KUKA KRL program: EPS_2_251806_MH58A_A_20260213065155.src

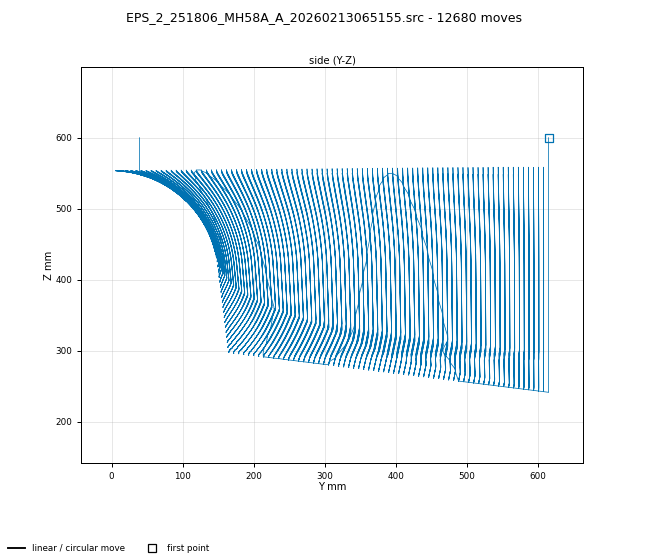
[picture p0: tool path of EPS_2_251806_MH58A_A_20260213065155.src, 12680 of 12682 moves have a stored position in this frame; points joined in program order, loops and branches not executed]
&ACCESS RVP
&REL 4
&COMMENT QRS 19112012
&PARAM EDITMASK = *
DEF PART()
EXT BAS (BAS_COMMAND :IN,REAL :IN )
INT I
BAS (#INITMOV,0 )

;KUKA QRS Post kuka4.cps  Date:22-06-2017 !

File_ID=3039

QRS_PRE_INIT()

;Init var - Until changes are made in qrs_pre_init
Outlet_Square_prg=0
Inlet_1_Square_prg=0
Inlet_2_Square_prg=0
Inlet_3_Square_prg=0
Inlet_4_Square_prg=0
Inlet_5_Square_prg=0

Outlet_1={X 0.000, Y 532.860, Z 433.000, B 0.000, E1 0.000 }
Inlet_1={X 0.000, Y 533.580, Z 423.000, B 0.000, E1 180.000 }
Outlet_1_type=251
Inlet_1_type=251
;QRS#1=Sidecore dimensions
;QRS#2=250-10" PVC SDR 35
;QRS#3=250-10" PVC SDR 35
;QRS#4=
;QRS#5=
;QRS#6=
;QRS#7=
;QRS#8=
;QRS#9=14M PSX
;QRS#10=14M PSX
;QRS#11=
;QRS#12=
;QRS#13=
;QRS#14=
;QRS#15=
;QRS#16=1220x127x838 2,75'
;QRS#17=EPS Height
;QRS#18=558,5
;QRS#19=*
;QRS#20= UPDATED VERSION 22-06-2017
;QRS#21=*
Outlet_Square=0100
Inlet_1_Square=0100
Inlet_2_Square=0
Inlet_3_Square=0
Inlet_4_Square=0
Inlet_5_Square=0
Mill_Square=1
Outlet_Square_Prg=205
Inlet_1_Square_prg=205

QRS_INIT()

$ADVANCE=5

; T1
PTP {E1 173.6,E2 173.6}
PTP {X 0,Y 615.5,A -85,B 0,C 180,E1 173.6,E2 173.6,E3 0,E4 0,E5 0,E6 0}
QRS_SPEED_INIT()
LIN {X 0,Y 615.5,Z 600,A -85,B 0,C 180,E1 173.6,E2 173.6,E3 0,E4 0,E5 0,E6 0} C_VEL
LIN {X 0,Y 615.5,Z 251.488,A -85,B 0,C 180,E1 173.6,E2 173.6} C_VEL
LIN {X 0,Y 615.5,Z 243.309,A -85,B 0,C 180,E1 173.6,E2 173.6} C_VEL
LIN {X 0,Y 615.485,Z 241.309,A -85,B 0,C 180,E1 173.413,E2 173.413} C_VEL
LIN {X 0,Y 615.489,Z 241.322,A -85,B 0,C 180,E1 170.801,E2 170.801} C_VEL
LIN {X 0,Y 615.477,Z 241.314,A -85,B 0,C 180,E1 168.139,E2 168.139} C_VEL
LIN {X 0,Y 615.482,Z 241.311,A -85,B 0,C 180,E1 165.451,E2 165.451} C_VEL
LIN {X 0,Y 615.491,Z 241.324,A -85,B 0,C 180,E1 162.73,E2 162.73} C_VEL
LIN {X 0,Y 615.489,Z 241.307,A -85,B 0,C 180,E1 159.967,E2 159.967} C_VEL
LIN {X 0,Y 615.482,Z 241.32,A -85,B 0,C 180,E1 157.155,E2 157.155} C_VEL
LIN {X 0,Y 615.476,Z 241.315,A -85,B 0,C 180,E1 154.431,E2 154.431} C_VEL
LIN {X 0,Y 615.483,Z 241.309,A -85,B 0,C 180,E1 152.085,E2 152.085} C_VEL
LIN {X 0,Y 615.488,Z 241.308,A -85,B 0,C 180,E1 149.84,E2 149.84} C_VEL
LIN {X 0,Y 615.478,Z 241.316,A -85,B 0,C 180,E1 147.542,E2 147.542} C_VEL
LIN {X 0,Y 615.494,Z 241.324,A -85,B 0,C 180,E1 145.185,E2 145.185} C_VEL
LIN {X 0,Y 615.476,Z 241.317,A -85,B 0,C 180,E1 142.757,E2 142.757} C_VEL
LIN {X 0,Y 615.484,Z 241.31,A -85,B 0,C 180,E1 139.91,E2 139.91} C_VEL
LIN {X 0,Y 615.481,Z 241.317,A -85,B 0,C 180,E1 137.646,E2 137.646} C_VEL
LIN {X 0,Y 615.477,Z 241.318,A -85,B 0,C 180,E1 134.93,E2 134.93} C_VEL
LIN {X 0,Y 615.486,Z 241.31,A -85,B 0,C 180,E1 132.08,E2 132.08} C_VEL
LIN {X 0,Y 615.482,Z 241.318,A -85,B 0,C 180,E1 129.75,E2 129.75} C_VEL
LIN {X 0,Y 615.474,Z 241.315,A -85,B 0,C 180,E1 126.935,E2 126.935} C_VEL
LIN {X 0,Y 615.48,Z 241.31,A -85,B 0,C 180,E1 124.699,E2 124.699} C_VEL
LIN {X 0,Y 615.491,Z 241.308,A -85,B 0,C 180,E1 122.331,E2 122.331} C_VEL
LIN {X 0,Y 615.485,Z 241.322,A -85,B 0,C 180,E1 119.406,E2 119.406} C_VEL
LIN {X 0,Y 615.473,Z 241.314,A -85,B 0,C 180,E1 117.042,E2 117.042} C_VEL
LIN {X 0,Y 615.483,Z 241.312,A -85,B 0,C 180,E1 114.272,E2 114.272} C_VEL
LIN {X 0,Y 615.493,Z 241.527,A -85,B 0,C 180,E1 111.651,E2 111.651} C_VEL
LIN {X 0,Y 615.453,Z 258.15,A -85,B 0,C 180,E1 109.339,E2 109.339} C_VEL
LIN {X 0,Y 615.483,Z 279.634,A -85,B 0,C 180,E1 106.429,E2 106.429} C_VEL
LIN {X 0,Y 615.481,Z 286.32,A -85,B 0,C 180,E1 105.565,E2 105.565} C_VEL
LIN {X 0,Y 615.477,Z 291.213,A -85,B 0,C 180,E1 105.48,E2 105.48} C_VEL
LIN {X 0,Y 615.499,Z 423.163,A -85,B 0,C 180,E1 103.905,E2 103.905} C_VEL
LIN {X 0,Y 615.497,Z 436.757,A -85,B 0,C 180,E1 103.621,E2 103.621} C_VEL
LIN {X 0,Y 615.498,Z 450.494,A -85,B 0,C 180,E1 103.201,E2 103.201} C_VEL
LIN {X 0,Y 615.492,Z 462.905,A -85,B 0,C 180,E1 102.697,E2 102.697} C_VEL
LIN {X 0,Y 615.486,Z 475.846,A -85,B 0,C 180,E1 102.028,E2 102.028} C_VEL
LIN {X 0,Y 615.499,Z 487.561,A -85,B 0,C 180,E1 101.276,E2 101.276} C_VEL
LIN {X 0,Y 615.498,Z 499.228,A -85,B 0,C 180,E1 100.36,E2 100.36} C_VEL
LIN {X 0,Y 615.497,Z 509.651,A -85,B 0,C 180,E1 99.364,E2 99.364} C_VEL
LIN {X 0,Y 615.496,Z 518.241,A -85,B 0,C 180,E1 98.371,E2 98.371} C_VEL
LIN {X 0,Y 615.495,Z 526.453,A -85,B 0,C 180,E1 97.215,E2 97.215} C_VEL
LIN {X 0,Y 615.496,Z 532.184,A -85,B 0,C 180,E1 96.227,E2 96.227} C_VEL
LIN {X 0,Y 615.494,Z 536.888,A -85,B 0,C 180,E1 95.241,E2 95.241} C_VEL
LIN {X 0,Y 615.496,Z 541.757,A -85,B 0,C 180,E1 93.928,E2 93.928} C_VEL
LIN {X 0,Y 615.496,Z 545.154,A -85,B 0,C 180,E1 92.618,E2 92.618} C_VEL
LIN {X 0,Y 615.493,Z 547.174,A -85,B 0,C 180,E1 91.309,E2 91.309} C_VEL
LIN {X 0,Y 615.494,Z 547.884,A -85,B 0,C 180,E1 90,E2 90} C_VEL
LIN {X 0,Y 615.49,Z 547.28,A -85,B 0,C 180,E1 88.691,E2 88.691} C_VEL
LIN {X 0,Y 615.493,Z 545.351,A -85,B 0,C 180,E1 87.382,E2 87.382} C_VEL
LIN {X 0,Y 615.496,Z 542.046,A -85,B 0,C 180,E1 86.072,E2 86.072} C_VEL
LIN {X 0,Y 615.496,Z 537.274,A -85,B 0,C 180,E1 84.759,E2 84.759} C_VEL
LIN {X 0,Y 615.494,Z 530.875,A -85,B 0,C 180,E1 83.444,E2 83.444} C_VEL
LIN {X 0,Y 615.496,Z 523.745,A -85,B 0,C 180,E1 82.29,E2 82.29} C_VEL
LIN {X 0,Y 615.497,Z 516.273,A -85,B 0,C 180,E1 81.298,E2 81.298} C_VEL
LIN {X 0,Y 615.496,Z 507.294,A -85,B 0,C 180,E1 80.304,E2 80.304} C_VEL
LIN {X 0,Y 615.499,Z 496.207,A -85,B 0,C 180,E1 79.291,E2 79.291} C_VEL
LIN {X 0,Y 615.498,Z 485.285,A -85,B 0,C 180,E1 78.474,E2 78.474} C_VEL
LIN {X 0,Y 615.486,Z 472.989,A -85,B 0,C 180,E1 77.721,E2 77.721} C_VEL
LIN {X 0,Y 615.494,Z 461.152,A -85,B 0,C 180,E1 77.135,E2 77.135} C_VEL
LIN {X 0,Y 615.495,Z 448.228,A -85,B 0,C 180,E1 76.631,E2 76.631} C_VEL
LIN {X 0,Y 615.498,Z 435.252,A -85,B 0,C 180,E1 76.253,E2 76.253} C_VEL
LIN {X 0,Y 615.497,Z 421.994,A -85,B 0,C 180,E1 75.988,E2 75.988} C_VEL
LIN {X 0,Y 615.477,Z 286.866,A -85,B 0,C 180,E1 74.371,E2 74.371} C_VEL
LIN {X 0,Y 615.483,Z 285.51,A -85,B 0,C 180,E1 74.265,E2 74.265} C_VEL
LIN {X 0,Y 615.476,Z 265.395,A -85,B 0,C 180,E1 71.558,E2 71.558} C_VEL
LIN {X 0,Y 615.499,Z 243.55,A -85,B 0,C 180,E1 68.569,E2 68.569} C_VEL
LIN {X 0,Y 615.497,Z 241.424,A -85,B 0,C 180,E1 68.217,E2 68.217} C_VEL
LIN {X 0,Y 615.486,Z 241.313,A -85,B 0,C 180,E1 65.729,E2 65.729} C_VEL
LIN {X 0,Y 615.468,Z 241.314,A -85,B 0,C 180,E1 62.959,E2 62.959} C_VEL
LIN {X 0,Y 615.491,Z 241.323,A -85,B 0,C 180,E1 60.205,E2 60.205} C_VEL
LIN {X 0,Y 615.493,Z 241.307,A -85,B 0,C 180,E1 57.544,E2 57.544} C_VEL
LIN {X 0,Y 615.473,Z 241.312,A -85,B 0,C 180,E1 55.185,E2 55.185} C_VEL
LIN {X 0,Y 615.477,Z 241.32,A -85,B 0,C 180,E1 52.758,E2 52.758} C_VEL
LIN {X 0,Y 615.484,Z 241.311,A -85,B 0,C 180,E1 49.912,E2 49.912} C_VEL
LIN {X 0,Y 615.495,Z 241.306,A -85,B 0,C 180,E1 47.649,E2 47.649} C_VEL
LIN {X 0,Y 615.475,Z 241.32,A -85,B 0,C 180,E1 44.932,E2 44.932} C_VEL
LIN {X 0,Y 615.485,Z 241.312,A -85,B 0,C 180,E1 42.081,E2 42.081} C_VEL
LIN {X 0,Y 615.489,Z 241.307,A -85,B 0,C 180,E1 39.75,E2 39.75} C_VEL
LIN {X 0,Y 615.477,Z 241.324,A -85,B 0,C 180,E1 36.937,E2 36.937} C_VEL
LIN {X 0,Y 615.488,Z 241.308,A -85,B 0,C 180,E1 34.022,E2 34.022} C_VEL
LIN {X 0,Y 615.48,Z 241.322,A -85,B 0,C 180,E1 31.087,E2 31.087} C_VEL
LIN {X 0,Y 615.482,Z 241.315,A -85,B 0,C 180,E1 28.452,E2 28.452} C_VEL
LIN {X 0,Y 615.476,Z 241.311,A -85,B 0,C 180,E1 25.716,E2 25.716} C_VEL
LIN {X 0,Y 615.473,Z 241.315,A -85,B 0,C 180,E1 23.557,E2 23.557} C_VEL
LIN {X 0,Y 615.476,Z 241.318,A -85,B 0,C 180,E1 21.432,E2 21.432} C_VEL
LIN {X 0,Y 615.481,Z 241.314,A -85,B 0,C 180,E1 18.607,E2 18.607} C_VEL
LIN {X 0,Y 615.477,Z 241.311,A -85,B 0,C 180,E1 15.906,E2 15.906} C_VEL
LIN {X 0,Y 615.497,Z 241.326,A -85,B 0,C 180,E1 13.201,E2 13.201} C_VEL
LIN {X 0,Y 615.487,Z 241.309,A -85,B 0,C 180,E1 10.527,E2 10.527} C_VEL
LIN {X 0,Y 615.475,Z 241.314,A -85,B 0,C 180,E1 7.876,E2 7.876} C_VEL
LIN {X 0,Y 615.491,Z 241.323,A -85,B 0,C 180,E1 5.241,E2 5.241} C_VEL
LIN {X 0,Y 615.489,Z 241.308,A -85,B 0,C 180,E1 2.618,E2 2.618} C_VEL
LIN {X 0,Y 615.476,Z 241.315,A -85,B 0,C 180,E1 0,E2 0} C_VEL
LIN {X 0,Y 615.49,Z 241.322,A -85,B 0,C 180,E1 -2.618,E2 -2.618} C_VEL
LIN {X 0,Y 615.488,Z 241.308,A -85,B 0,C 180,E1 -5.241,E2 -5.241} C_VEL
LIN {X 0,Y 615.477,Z 241.315,A -85,B 0,C 180,E1 -7.876,E2 -7.876} C_VEL
LIN {X 0,Y 615.487,Z 241.321,A -85,B 0,C 180,E1 -10.527,E2 -10.527} C_VEL
LIN {X 0,Y 615.494,Z 241.306,A -85,B 0,C 180,E1 -13.201,E2 -13.201} C_VEL
LIN {X 0,Y 615.477,Z 241.319,A -85,B 0,C 180,E1 -15.905,E2 -15.905} C_VEL
LIN {X 0,Y 615.476,Z 241.316,A -85,B 0,C 180,E1 -18.646,E2 -18.646} C_VEL
LIN {X 0,Y 615.479,Z 241.311,A -85,B 0,C 180,E1 -21.432,E2 -21.432} C_VEL
LIN {X 0,Y 615.482,Z 241.322,A -85,B 0,C 180,E1 -24.272,E2 -24.272} C_VEL
LIN {X 0,Y 615.49,Z 241.307,A -85,B 0,C 180,E1 -27.177,E2 -27.177} C_VEL
LIN {X 0,Y 615.486,Z 241.321,A -85,B 0,C 180,E1 -30.16,E2 -30.16} C_VEL
LIN {X 0,Y 615.473,Z 241.315,A -85,B 0,C 180,E1 -32.458,E2 -32.458} C_VEL
LIN {X 0,Y 615.49,Z 241.307,A -85,B 0,C 180,E1 -34.815,E2 -34.815} C_VEL
LIN {X 0,Y 615.481,Z 241.313,A -85,B 0,C 180,E1 -37.243,E2 -37.243} C_VEL
LIN {X 0,Y 615.479,Z 241.319,A -85,B 0,C 180,E1 -40.09,E2 -40.09} C_VEL
LIN {X 0,Y 615.475,Z 241.313,A -85,B 0,C 180,E1 -42.354,E2 -42.354} C_VEL
LIN {X 0,Y 615.482,Z 241.312,A -85,B 0,C 180,E1 -45.069,E2 -45.069} C_VEL
LIN {X 0,Y 615.48,Z 241.32,A -85,B 0,C 180,E1 -47.921,E2 -47.921} C_VEL
LIN {X 0,Y 615.475,Z 241.313,A -85,B 0,C 180,E1 -50.25,E2 -50.25} C_VEL
LIN {X 0,Y 615.479,Z 241.315,A -85,B 0,C 180,E1 -53.065,E2 -53.065} C_VEL
LIN {X 0,Y 615.488,Z 241.321,A -85,B 0,C 180,E1 -55.299,E2 -55.299} C_VEL
LIN {X 0,Y 615.483,Z 241.321,A -85,B 0,C 180,E1 -57.67,E2 -57.67} C_VEL
LIN {X 0,Y 615.493,Z 241.307,A -85,B 0,C 180,E1 -60.595,E2 -60.595} C_VEL
LIN {X 0,Y 615.481,Z 241.322,A -85,B 0,C 180,E1 -63.556,E2 -63.556} C_VEL
LIN {X 0,Y 615.486,Z 241.308,A -85,B 0,C 180,E1 -66.444,E2 -66.444} C_VEL
LIN {X 0,Y 615.497,Z 241.502,A -85,B 0,C 180,E1 -67.343,E2 -67.343} C_VEL
LIN {X 0,Y 615.494,Z 249.16,A -85,B 0,C 180,E1 -68.393,E2 -68.393} C_VEL
LIN {X 0,Y 615.433,Z 270.63,A -85,B 0,C 180,E1 -71.18,E2 -71.18} C_VEL
LIN {X 0,Y 615.481,Z 291.387,A -85,B 0,C 180,E1 -73.838,E2 -73.838} C_VEL
LIN {X 0,Y 615.49,Z 296.026,A -85,B 0,C 180,E1 -74.393,E2 -74.393} C_VEL
LIN {X 0,Y 615.479,Z 315.746,A -85,B 0,C 180,E1 -74.647,E2 -74.647} C_VEL
LIN {X 0,Y 615.5,Z 433.901,A -85,B 0,C 180,E1 -76.063,E2 -76.063} C_VEL
LIN {X 0,Y 615.497,Z 448.389,A -85,B 0,C 180,E1 -76.379,E2 -76.379} C_VEL
LIN {X 0,Y 615.496,Z 461.697,A -85,B 0,C 180,E1 -76.799,E2 -76.799} C_VEL
LIN {X 0,Y 615.497,Z 473.843,A -85,B 0,C 180,E1 -77.303,E2 -77.303} C_VEL
LIN {X 0,Y 615.485,Z 486.605,A -85,B 0,C 180,E1 -77.972,E2 -77.972} C_VEL
LIN {X 0,Y 615.499,Z 499.344,A -85,B 0,C 180,E1 -78.807,E2 -78.807} C_VEL
LIN {X 0,Y 615.498,Z 509.751,A -85,B 0,C 180,E1 -79.64,E2 -79.64} C_VEL
LIN {X 0,Y 615.496,Z 520.09,A -85,B 0,C 180,E1 -80.636,E2 -80.636} C_VEL
LIN {X 0,Y 615.497,Z 528.604,A -85,B 0,C 180,E1 -81.629,E2 -81.629} C_VEL
LIN {X 0,Y 615.496,Z 536.728,A -85,B 0,C 180,E1 -82.785,E2 -82.785} C_VEL
LIN {X 0,Y 615.496,Z 542.431,A -85,B 0,C 180,E1 -83.773,E2 -83.773} C_VEL
LIN {X 0,Y 615.495,Z 547.081,A -85,B 0,C 180,E1 -84.759,E2 -84.759} C_VEL
LIN {X 0,Y 615.494,Z 551.902,A -85,B 0,C 180,E1 -86.072,E2 -86.072} C_VEL
LIN {X 0,Y 615.496,Z 555.252,A -85,B 0,C 180,E1 -87.382,E2 -87.382} C_VEL
LIN {X 0,Y 615.489,Z 557.229,A -85,B 0,C 180,E1 -88.691,E2 -88.691} C_VEL
LIN {X 0,Y 615.493,Z 557.889,A -85,B 0,C 180,E1 -90,E2 -90} C_VEL
LIN {X 0,Y 615.489,Z 557.229,A -85,B 0,C 180,E1 -91.309,E2 -91.309} C_VEL
LIN {X 0,Y 615.496,Z 555.252,A -85,B 0,C 180,E1 -92.618,E2 -92.618} C_VEL
LIN {X 0,Y 615.494,Z 551.902,A -85,B 0,C 180,E1 -93.928,E2 -93.928} C_VEL
LIN {X 0,Y 615.495,Z 547.081,A -85,B 0,C 180,E1 -95.241,E2 -95.241} C_VEL
LIN {X 0,Y 615.496,Z 540.628,A -85,B 0,C 180,E1 -96.556,E2 -96.556} C_VEL
LIN {X 0,Y 615.497,Z 533.441,A -85,B 0,C 180,E1 -97.71,E2 -97.71} C_VEL
LIN {X 0,Y 615.498,Z 525.904,A -85,B 0,C 180,E1 -98.702,E2 -98.702} C_VEL
LIN {X 0,Y 615.496,Z 516.854,A -85,B 0,C 180,E1 -99.696,E2 -99.696} C_VEL
LIN {X 0,Y 615.498,Z 506.758,A -85,B 0,C 180,E1 -100.618,E2 -100.618} C_VEL
LIN {X 0,Y 615.498,Z 495.86,A -85,B 0,C 180,E1 -101.443,E2 -101.443} C_VEL
LIN {X 0,Y 615.485,Z 483.71,A -85,B 0,C 180,E1 -102.195,E2 -102.195} C_VEL
LIN {X 0,Y 615.495,Z 470.095,A -85,B 0,C 180,E1 -102.865,E2 -102.865} C_VEL
LIN {X 0,Y 615.496,Z 456.841,A -85,B 0,C 180,E1 -103.369,E2 -103.369} C_VEL
LIN {X 0,Y 615.498,Z 443.296,A -85,B 0,C 180,E1 -103.747,E2 -103.747} C_VEL
LIN {X 0,Y 615.497,Z 428.756,A -85,B 0,C 180,E1 -104.013,E2 -104.013} C_VEL
LIN {X 0,Y 615.488,Z 296.53,A -85,B 0,C 180,E1 -105.586,E2 -105.586} C_VEL
LIN {X 0,Y 615.493,Z 295.48,A -85,B 0,C 180,E1 -105.65,E2 -105.65} C_VEL
LIN {X 0,Y 615.435,Z 273.652,A -85,B 0,C 180,E1 -108.431,E2 -108.431} C_VEL
LIN {X 0,Y 615.46,Z 254.529,A -85,B 0,C 180,E1 -110.906,E2 -110.906} C_VEL
LIN {X 0,Y 615.497,Z 241.605,A -85,B 0,C 180,E1 -112.626,E2 -112.626} C_VEL
LIN {X 0,Y 615.492,Z 241.323,A -85,B 0,C 180,E1 -112.844,E2 -112.844} C_VEL
LIN {X 0,Y 615.485,Z 241.308,A -85,B 0,C 180,E1 -115.715,E2 -115.715} C_VEL
LIN {X 0,Y 615.486,Z 241.327,A -85,B 0,C 180,E1 -118.657,E2 -118.657} C_VEL
LIN {X 0,Y 615.482,Z 241.314,A -85,B 0,C 180,E1 -121.085,E2 -121.085} C_VEL
LIN {X 0,Y 615.492,Z 241.307,A -85,B 0,C 180,E1 -123.535,E2 -123.535} C_VEL
LIN {X 0,Y 615.482,Z 241.327,A -85,B 0,C 180,E1 -126.424,E2 -126.424} C_VEL
LIN {X 0,Y 615.484,Z 241.311,A -85,B 0,C 180,E1 -129.062,E2 -129.062} C_VEL
LIN {X 0,Y 615.486,Z 241.308,A -85,B 0,C 180,E1 -131.473,E2 -131.473} C_VEL
LIN {X 0,Y 615.485,Z 241.321,A -85,B 0,C 180,E1 -134.149,E2 -134.149} C_VEL
LIN {X 0,Y 615.484,Z 241.311,A -85,B 0,C 180,E1 -136.952,E2 -136.952} C_VEL
LIN {X 0,Y 615.48,Z 241.31,A -85,B 0,C 180,E1 -139.393,E2 -139.393} C_VEL
LIN {X 0,Y 615.483,Z 241.321,A -85,B 0,C 180,E1 -141.987,E2 -141.987} C_VEL
LIN {X 0,Y 615.486,Z 241.32,A -85,B 0,C 180,E1 -144.384,E2 -144.384} C_VEL
LIN {X 0,Y 615.483,Z 241.311,A -85,B 0,C 180,E1 -146.763,E2 -146.763} C_VEL
LIN {X 0,Y 615.486,Z 241.308,A -85,B 0,C 180,E1 -149.08,E2 -149.08} C_VEL
LIN {X 0,Y 615.475,Z 241.316,A -85,B 0,C 180,E1 -151.55,E2 -151.55} C_VEL
LIN {X 0,Y 615.482,Z 241.319,A -85,B 0,C 180,E1 -154.284,E2 -154.284} C_VEL
LIN {X 0,Y 615.478,Z 241.315,A -85,B 0,C 180,E1 -156.443,E2 -156.443} C_VEL
LIN {X 0,Y 615.479,Z 241.312,A -85,B 0,C 180,E1 -158.568,E2 -158.568} C_VEL
LIN {X 0,Y 615.475,Z 241.316,A -85,B 0,C 180,E1 -161.354,E2 -161.354} C_VEL
LIN {X 0,Y 615.482,Z 241.319,A -85,B 0,C 180,E1 -164.095,E2 -164.095} C_VEL
LIN {X 0,Y 615.493,Z 241.306,A -85,B 0,C 180,E1 -166.799,E2 -166.799} C_VEL
LIN {X 0,Y 615.484,Z 241.321,A -85,B 0,C 180,E1 -169.473,E2 -169.473} C_VEL
LIN {X 0,Y 615.478,Z 241.315,A -85,B 0,C 180,E1 -172.124,E2 -172.124} C_VEL
LIN {X 0,Y 615.487,Z 241.308,A -85,B 0,C 180,E1 -174.759,E2 -174.759} C_VEL
LIN {X 0,Y 615.487,Z 241.322,A -85,B 0,C 180,E1 -177.382,E2 -177.382} C_VEL
LIN {X 0,Y 615.478,Z 241.315,A -85,B 0,C 180,E1 -180,E2 -180} C_VEL
LIN {X 0,Y 615.488,Z 241.308,A -85,B 0,C 180,E1 -182.618,E2 -182.618} C_VEL
LIN {X 0,Y 615.487,Z 241.322,A -85,B 0,C 180,E1 -185.241,E2 -185.241} C_VEL
LIN {X 0,Y 615.485,Z 241.309,A -85,B 0,C 180,E1 -186.587,E2 -186.587} C_VEL
LIN {X 0,Y 614.81,Z 241.47,A -85,B 0,C 180,E1 -187.133,E2 -187.133} C_VEL
LIN {X 0,Y 611.978,Z 241.874,A -85,B 0,C 180,E1 -188.019,E2 -188.019} C_VEL
LIN {X 0,Y 609.586,Z 242.191,A -85,B 0,C 180,E1 -188.731,E2 -188.731} C_VEL
LIN {X 0,Y 608.548,Z 242.311,A -85,B 0,C 180,E1 -189.281,E2 -189.281} C_VEL
LIN {X 0,Y 608.457,Z 242.319,A -85,B 0,C 180,E1 -189.467,E2 -189.467} C_VEL
LIN {X 0,Y 608.454,Z 242.313,A -85,B 0,C 180,E1 -192,E2 -192} C_VEL
LIN {X 0,Y 608.472,Z 242.312,A -85,B 0,C 180,E1 -194.721,E2 -194.721} C_VEL
LIN {X 0,Y 608.453,Z 242.318,A -85,B 0,C 180,E1 -197.477,E2 -197.477} C_VEL
LIN {X 0,Y 608.46,Z 242.311,A -85,B 0,C 180,E1 -200.274,E2 -200.274} C_VEL
LIN {X 0,Y 608.449,Z 242.314,A -85,B 0,C 180,E1 -202.477,E2 -202.477} C_VEL
LIN {X 0,Y 608.456,Z 242.315,A -85,B 0,C 180,E1 -204.571,E2 -204.571} C_VEL
LIN {X 0,Y 608.48,Z 242.316,A -85,B 0,C 180,E1 -207.21,E2 -207.21} C_VEL
LIN {X 0,Y 608.466,Z 242.311,A -85,B 0,C 180,E1 -209.973,E2 -209.973} C_VEL
LIN {X 0,Y 608.454,Z 242.316,A -85,B 0,C 180,E1 -212.523,E2 -212.523} C_VEL
LIN {X 0,Y 608.442,Z 242.317,A -85,B 0,C 180,E1 -215.278,E2 -215.278} C_VEL
LIN {X 0,Y 608.465,Z 242.311,A -85,B 0,C 180,E1 -217.747,E2 -217.747} C_VEL
LIN {X 0,Y 608.449,Z 242.316,A -85,B 0,C 180,E1 -220.33,E2 -220.33} C_VEL
LIN {X 0,Y 608.446,Z 242.32,A -85,B 0,C 180,E1 -222.961,E2 -222.961} C_VEL
LIN {X 0,Y 608.459,Z 242.312,A -85,B 0,C 180,E1 -225.736,E2 -225.736} C_VEL
LIN {X 0,Y 608.463,Z 242.321,A -85,B 0,C 180,E1 -228.658,E2 -228.658} C_VEL
LIN {X 0,Y 608.461,Z 242.311,A -85,B 0,C 180,E1 -231.412,E2 -231.412} C_VEL
LIN {X 0,Y 608.475,Z 242.312,A -85,B 0,C 180,E1 -233.951,E2 -233.951} C_VEL
LIN {X 0,Y 608.469,Z 242.318,A -85,B 0,C 180,E1 -236.33,E2 -236.33} C_VEL
LIN {X 0,Y 608.444,Z 242.319,A -85,B 0,C 180,E1 -238.733,E2 -238.733} C_VEL
LIN {X 0,Y 608.473,Z 242.31,A -85,B 0,C 180,E1 -241.381,E2 -241.381} C_VEL
LIN {X 0,Y 608.478,Z 242.319,A -85,B 0,C 180,E1 -244.278,E2 -244.278} C_VEL
LIN {X 0,Y 608.446,Z 242.316,A -85,B 0,C 180,E1 -246.876,E2 -246.876} C_VEL
LIN {X 0,Y 608.512,Z 242.509,A -85,B 0,C 180,E1 -248.244,E2 -248.244} C_VEL
LIN {X 0,Y 608.516,Z 258.17,A -85,B 0,C 180,E1 -250.432,E2 -250.432} C_VEL
LIN {X 0,Y 608.527,Z 278.525,A -85,B 0,C 180,E1 -253.218,E2 -253.218} C_VEL
LIN {X 0,Y 608.535,Z 286.323,A -85,B 0,C 180,E1 -254.253,E2 -254.253} C_VEL
LIN {X 0,Y 608.651,Z 289.47,A -85,B 0,C 180,E1 -254.32,E2 -254.32} C_VEL
LIN {X 0,Y 608.608,Z 423.991,A -85,B 0,C 180,E1 -255.949,E2 -255.949} C_VEL
LIN {X 0,Y 608.613,Z 438.305,A -85,B 0,C 180,E1 -256.264,E2 -256.264} C_VEL
LIN {X 0,Y 608.586,Z 451.65,A -85,B 0,C 180,E1 -256.689,E2 -256.689} C_VEL
LIN {X 0,Y 608.542,Z 464.709,A -85,B 0,C 180,E1 -257.24,E2 -257.24} C_VEL
LIN {X 0,Y 608.529,Z 477.345,A -85,B 0,C 180,E1 -257.917,E2 -257.917} C_VEL
LIN {X 0,Y 608.499,Z 488.854,A -85,B 0,C 180,E1 -258.677,E2 -258.677} C_VEL
LIN {X 0,Y 608.495,Z 499.414,A -85,B 0,C 180,E1 -259.519,E2 -259.519} C_VEL
LIN {X 0,Y 608.48,Z 509.9,A -85,B 0,C 180,E1 -260.527,E2 -260.527} C_VEL
LIN {X 0,Y 608.463,Z 518.552,A -85,B 0,C 180,E1 -261.532,E2 -261.532} C_VEL
LIN {X 0,Y 608.46,Z 526.84,A -85,B 0,C 180,E1 -262.701,E2 -262.701} C_VEL
LIN {X 0,Y 608.443,Z 533.325,A -85,B 0,C 180,E1 -263.831,E2 -263.831} C_VEL
LIN {X 0,Y 608.435,Z 538.788,A -85,B 0,C 180,E1 -265.03,E2 -265.03} C_VEL
LIN {X 0,Y 608.434,Z 542.298,A -85,B 0,C 180,E1 -266.026,E2 -266.026} C_VEL
LIN {X 0,Y 608.424,Z 545.734,A -85,B 0,C 180,E1 -267.352,E2 -267.352} C_VEL
LIN {X 0,Y 608.446,Z 547.777,A -85,B 0,C 180,E1 -268.676,E2 -268.676} C_VEL
LIN {X 0,Y 608.434,Z 548.495,A -85,B 0,C 180,E1 -270,E2 -270} C_VEL
LIN {X 0,Y 608.443,Z 547.882,A -85,B 0,C 180,E1 -271.324,E2 -271.324} C_VEL
LIN {X 0,Y 608.421,Z 545.928,A -85,B 0,C 180,E1 -272.648,E2 -272.648} C_VEL
LIN {X 0,Y 608.434,Z 542.585,A -85,B 0,C 180,E1 -273.974,E2 -273.974} C_VEL
LIN {X 0,Y 608.44,Z 537.761,A -85,B 0,C 180,E1 -275.302,E2 -275.302} C_VEL
LIN {X 0,Y 608.442,Z 531.474,A -85,B 0,C 180,E1 -276.6,E2 -276.6} C_VEL
LIN {X 0,Y 608.453,Z 524.101,A -85,B 0,C 180,E1 -277.8,E2 -277.8} C_VEL
LIN {X 0,Y 608.476,Z 516.565,A -85,B 0,C 180,E1 -278.803,E2 -278.803} C_VEL
LIN {X 0,Y 608.488,Z 507.52,A -85,B 0,C 180,E1 -279.809,E2 -279.809} C_VEL
LIN {X 0,Y 608.507,Z 496.723,A -85,B 0,C 180,E1 -280.804,E2 -280.804} C_VEL
LIN {X 0,Y 608.523,Z 485.387,A -85,B 0,C 180,E1 -281.66,E2 -281.66} C_VEL
LIN {X 0,Y 608.539,Z 473.045,A -85,B 0,C 180,E1 -282.421,E2 -282.421} C_VEL
LIN {X 0,Y 608.559,Z 461.177,A -85,B 0,C 180,E1 -283.014,E2 -283.014} C_VEL
LIN {X 0,Y 608.581,Z 448.228,A -85,B 0,C 180,E1 -283.524,E2 -283.524} C_VEL
LIN {X 0,Y 608.594,Z 433.992,A -85,B 0,C 180,E1 -283.935,E2 -283.935} C_VEL
LIN {X 0,Y 608.624,Z 419.126,A -85,B 0,C 180,E1 -284.214,E2 -284.214} C_VEL
LIN {X 0,Y 608.565,Z 286.83,A -85,B 0,C 180,E1 -285.811,E2 -285.811} C_VEL
LIN {X 0,Y 608.493,Z 285.56,A -85,B 0,C 180,E1 -285.92,E2 -285.92} C_VEL
LIN {X 0,Y 608.503,Z 266.614,A -85,B 0,C 180,E1 -288.497,E2 -288.497} C_VEL
LIN {X 0,Y 608.579,Z 244.822,A -85,B 0,C 180,E1 -291.509,E2 -291.509} C_VEL
LIN {X 0,Y 608.479,Z 242.468,A -85,B 0,C 180,E1 -291.869,E2 -291.869} C_VEL
LIN {X 0,Y 608.448,Z 242.313,A -85,B 0,C 180,E1 -294.571,E2 -294.571} C_VEL
LIN {X 0,Y 608.464,Z 242.314,A -85,B 0,C 180,E1 -297.204,E2 -297.204} C_VEL
LIN {X 0,Y 608.469,Z 242.316,A -85,B 0,C 180,E1 -299.971,E2 -299.971} C_VEL
LIN {X 0,Y 608.454,Z 242.313,A -85,B 0,C 180,E1 -302.879,E2 -302.879} C_VEL
LIN {X 0,Y 608.441,Z 242.319,A -85,B 0,C 180,E1 -305.277,E2 -305.277} C_VEL
LIN {X 0,Y 608.464,Z 242.312,A -85,B 0,C 180,E1 -308.24,E2 -308.24} C_VEL
LIN {X 0,Y 608.447,Z 242.313,A -85,B 0,C 180,E1 -310.328,E2 -310.328} C_VEL
LIN {X 0,Y 608.443,Z 242.316,A -85,B 0,C 180,E1 -312.959,E2 -312.959} C_VEL
LIN {X 0,Y 608.452,Z 242.317,A -85,B 0,C 180,E1 -315.735,E2 -315.735} C_VEL
LIN {X 0,Y 608.451,Z 242.313,A -85,B 0,C 180,E1 -318.657,E2 -318.657} C_VEL
LIN {X 0,Y 608.466,Z 242.319,A -85,B 0,C 180,E1 -321.412,E2 -321.412} C_VEL
LIN {X 0,Y 608.474,Z 242.31,A -85,B 0,C 180,E1 -323.949,E2 -323.949} C_VEL
LIN {X 0,Y 608.456,Z 242.312,A -85,B 0,C 180,E1 -326.329,E2 -326.329} C_VEL
LIN {X 0,Y 608.47,Z 242.314,A -85,B 0,C 180,E1 -328.727,E2 -328.727} C_VEL
LIN {X 0,Y 608.47,Z 242.316,A -85,B 0,C 180,E1 -331.378,E2 -331.378} C_VEL
LIN {X 0,Y 608.438,Z 242.314,A -85,B 0,C 180,E1 -333.964,E2 -333.964} C_VEL
LIN {X 0,Y 608.466,Z 242.311,A -85,B 0,C 180,E1 -336.155,E2 -336.155} C_VEL
LIN {X 0,Y 608.449,Z 242.322,A -85,B 0,C 180,E1 -339.018,E2 -339.018} C_VEL
LIN {X 0,Y 608.444,Z 242.313,A -85,B 0,C 180,E1 -341.828,E2 -341.828} C_VEL
LIN {X 0,Y 608.471,Z 242.316,A -85,B 0,C 180,E1 -344.594,E2 -344.594} C_VEL
LIN {X 0,Y 608.476,Z 242.312,A -85,B 0,C 180,E1 -347.323,E2 -347.323} C_VEL
LIN {X 0,Y 608.447,Z 242.314,A -85,B 0,C 180,E1 -350.022,E2 -350.022} C_VEL
LIN {X 0,Y 608.478,Z 242.32,A -85,B 0,C 180,E1 -352.701,E2 -352.701} C_VEL
LIN {X 0,Y 608.455,Z 242.313,A -85,B 0,C 180,E1 -355.362,E2 -355.362} C_VEL
LIN {X 0,Y 608.446,Z 242.315,A -85,B 0,C 180,E1 -358.014,E2 -358.014} C_VEL
LIN {X 0,Y 608.479,Z 242.317,A -85,B 0,C 180,E1 -360.662,E2 -360.662} C_VEL
LIN {X 0,Y 608.476,Z 242.31,A -85,B 0,C 180,E1 -363.311,E2 -363.311} C_VEL
LIN {X 0,Y 608.451,Z 242.316,A -85,B 0,C 180,E1 -365.967,E2 -365.967} C_VEL
LIN {X 0,Y 608.455,Z 242.318,A -85,B 0,C 180,E1 -368.636,E2 -368.636} C_VEL
LIN {X 0,Y 608.472,Z 242.31,A -85,B 0,C 180,E1 -371.324,E2 -371.324} C_VEL
LIN {X 0,Y 608.458,Z 242.318,A -85,B 0,C 180,E1 -374.038,E2 -374.038} C_VEL
LIN {X 0,Y 608.47,Z 242.312,A -85,B 0,C 180,E1 -376.784,E2 -376.784} C_VEL
LIN {X 0,Y 608.453,Z 242.314,A -85,B 0,C 180,E1 -379.571,E2 -379.571} C_VEL
LIN {X 0,Y 608.448,Z 242.317,A -85,B 0,C 180,E1 -382.477,E2 -382.477} C_VEL
LIN {X 0,Y 608.452,Z 242.315,A -85,B 0,C 180,E1 -384.571,E2 -384.571} C_VEL
LIN {X 0,Y 608.482,Z 242.309,A -85,B 0,C 180,E1 -387.21,E2 -387.21} C_VEL
LIN {X 0,Y 608.467,Z 242.322,A -85,B 0,C 180,E1 -389.974,E2 -389.974} C_VEL
LIN {X 0,Y 608.449,Z 242.314,A -85,B 0,C 180,E1 -392.523,E2 -392.523} C_VEL
LIN {X 0,Y 608.443,Z 242.315,A -85,B 0,C 180,E1 -395.278,E2 -395.278} C_VEL
LIN {X 0,Y 608.465,Z 242.32,A -85,B 0,C 180,E1 -397.747,E2 -397.747} C_VEL
LIN {X 0,Y 608.445,Z 242.315,A -85,B 0,C 180,E1 -400.33,E2 -400.33} C_VEL
LIN {X 0,Y 608.468,Z 242.314,A -85,B 0,C 180,E1 -403.31,E2 -403.31} C_VEL
LIN {X 0,Y 608.465,Z 242.314,A -85,B 0,C 180,E1 -406.131,E2 -406.131} C_VEL
LIN {X 0,Y 608.456,Z 242.312,A -85,B 0,C 180,E1 -408.825,E2 -408.825} C_VEL
LIN {X 0,Y 608.463,Z 242.319,A -85,B 0,C 180,E1 -411.413,E2 -411.413} C_VEL
LIN {X 0,Y 608.442,Z 242.317,A -85,B 0,C 180,E1 -413.955,E2 -413.955} C_VEL
LIN {X 0,Y 608.464,Z 242.311,A -85,B 0,C 180,E1 -416.33,E2 -416.33} C_VEL
LIN {X 0,Y 608.475,Z 242.311,A -85,B 0,C 180,E1 -418.728,E2 -418.728} C_VEL
LIN {X 0,Y 608.472,Z 242.321,A -85,B 0,C 180,E1 -421.38,E2 -421.38} C_VEL
LIN {X 0,Y 608.474,Z 242.31,A -85,B 0,C 180,E1 -424.279,E2 -424.279} C_VEL
LIN {X 0,Y 608.5,Z 242.427,A -85,B 0,C 180,E1 -427.193,E2 -427.193} C_VEL
LIN {X 0,Y 608.596,Z 245.132,A -85,B 0,C 180,E1 -427.6,E2 -427.6} C_VEL
LIN {X 0,Y 608.545,Z 267.959,A -85,B 0,C 180,E1 -430.608,E2 -430.608} C_VEL
LIN {X 0,Y 608.453,Z 288.1,A -85,B 0,C 180,E1 -433.216,E2 -433.216} C_VEL
LIN {X 0,Y 608.551,Z 296.02,A -85,B 0,C 180,E1 -434.21,E2 -434.21} C_VEL
LIN {X 0,Y 608.669,Z 299.648,A -85,B 0,C 180,E1 -434.278,E2 -434.278} C_VEL
LIN {X 0,Y 608.621,Z 432.931,A -85,B 0,C 180,E1 -435.885,E2 -435.885} C_VEL
LIN {X 0,Y 608.607,Z 446.874,A -85,B 0,C 180,E1 -436.179,E2 -436.179} C_VEL
LIN {X 0,Y 608.565,Z 460.597,A -85,B 0,C 180,E1 -436.604,E2 -436.604} C_VEL
LIN {X 0,Y 608.562,Z 473.889,A -85,B 0,C 180,E1 -437.156,E2 -437.156} C_VEL
LIN {X 0,Y 608.513,Z 486.685,A -85,B 0,C 180,E1 -437.832,E2 -437.832} C_VEL
LIN {X 0,Y 608.499,Z 499.474,A -85,B 0,C 180,E1 -438.677,E2 -438.677} C_VEL
LIN {X 0,Y 608.496,Z 509.934,A -85,B 0,C 180,E1 -439.519,E2 -439.519} C_VEL
LIN {X 0,Y 608.479,Z 520.336,A -85,B 0,C 180,E1 -440.527,E2 -440.527} C_VEL
LIN {X 0,Y 608.464,Z 528.916,A -85,B 0,C 180,E1 -441.532,E2 -441.532} C_VEL
LIN {X 0,Y 608.461,Z 537.115,A -85,B 0,C 180,E1 -442.701,E2 -442.701} C_VEL
LIN {X 0,Y 608.444,Z 543.546,A -85,B 0,C 180,E1 -443.831,E2 -443.831} C_VEL
LIN {X 0,Y 608.437,Z 548.962,A -85,B 0,C 180,E1 -445.03,E2 -445.03} C_VEL
LIN {X 0,Y 608.431,Z 552.442,A -85,B 0,C 180,E1 -446.026,E2 -446.026} C_VEL
LIN {X 0,Y 608.424,Z 555.831,A -85,B 0,C 180,E1 -447.352,E2 -447.352} C_VEL
LIN {X 0,Y 608.442,Z 557.83,A -85,B 0,C 180,E1 -448.676,E2 -448.676} C_VEL
LIN {X 0,Y 608.433,Z 558.5,A -85,B 0,C 180,E1 -450,E2 -450} C_VEL
LIN {X 0,Y 608.442,Z 557.83,A -85,B 0,C 180,E1 -451.324,E2 -451.324} C_VEL
LIN {X 0,Y 608.424,Z 555.831,A -85,B 0,C 180,E1 -452.648,E2 -452.648} C_VEL
LIN {X 0,Y 608.431,Z 552.441,A -85,B 0,C 180,E1 -453.974,E2 -453.974} C_VEL
LIN {X 0,Y 608.44,Z 547.568,A -85,B 0,C 180,E1 -455.302,E2 -455.302} C_VEL
LIN {X 0,Y 608.445,Z 541.212,A -85,B 0,C 180,E1 -456.603,E2 -456.603} C_VEL
LIN {X 0,Y 608.453,Z 533.798,A -85,B 0,C 180,E1 -457.8,E2 -457.8} C_VEL
LIN {X 0,Y 608.473,Z 524.824,A -85,B 0,C 180,E1 -458.97,E2 -458.97} C_VEL
LIN {X 0,Y 608.473,Z 515.392,A -85,B 0,C 180,E1 -459.977,E2 -459.977} C_VEL
LIN {X 0,Y 608.506,Z 504.047,A -85,B 0,C 180,E1 -460.973,E2 -460.973} C_VEL
LIN {X 0,Y 608.531,Z 492.151,A -85,B 0,C 180,E1 -461.829,E2 -461.829} C_VEL
LIN {X 0,Y 608.529,Z 479.076,A -85,B 0,C 180,E1 -462.591,E2 -462.591} C_VEL
LIN {X 0,Y 608.561,Z 466.177,A -85,B 0,C 180,E1 -463.184,E2 -463.184} C_VEL
LIN {X 0,Y 608.596,Z 452.189,A -85,B 0,C 180,E1 -463.672,E2 -463.672} C_VEL
LIN {X 0,Y 608.621,Z 438.464,A -85,B 0,C 180,E1 -464.012,E2 -464.012} C_VEL
LIN {X 0,Y 608.627,Z 422.183,A -85,B 0,C 180,E1 -464.257,E2 -464.257} C_VEL
LIN {X 0,Y 608.604,Z 296.517,A -85,B 0,C 180,E1 -465.767,E2 -465.767} C_VEL
LIN {X 0,Y 608.521,Z 295.525,A -85,B 0,C 180,E1 -465.834,E2 -465.834} C_VEL
LIN {X 0,Y 608.48,Z 274.9,A -85,B 0,C 180,E1 -468.489,E2 -468.489} C_VEL
LIN {X 0,Y 608.518,Z 257.4,A -85,B 0,C 180,E1 -470.778,E2 -470.778} C_VEL
LIN {X 0,Y 608.561,Z 242.969,A -85,B 0,C 180,E1 -472.697,E2 -472.697} C_VEL
LIN {X 0,Y 608.487,Z 242.382,A -85,B 0,C 180,E1 -472.852,E2 -472.852} C_VEL
LIN {X 0,Y 608.474,Z 242.31,A -85,B 0,C 180,E1 -475.721,E2 -475.721} C_VEL
LIN {X 0,Y 608.472,Z 242.321,A -85,B 0,C 180,E1 -478.62,E2 -478.62} C_VEL
LIN {X 0,Y 608.458,Z 242.313,A -85,B 0,C 180,E1 -481.316,E2 -481.316} C_VEL
LIN {X 0,Y 608.472,Z 242.31,A -85,B 0,C 180,E1 -483.735,E2 -483.735} C_VEL
LIN {X 0,Y 608.442,Z 242.318,A -85,B 0,C 180,E1 -486.092,E2 -486.092} C_VEL
LIN {X 0,Y 608.463,Z 242.319,A -85,B 0,C 180,E1 -488.587,E2 -488.587} C_VEL
LIN {X 0,Y 608.462,Z 242.311,A -85,B 0,C 180,E1 -491.342,E2 -491.342} C_VEL
LIN {X 0,Y 608.453,Z 242.322,A -85,B 0,C 180,E1 -494.264,E2 -494.264} C_VEL
LIN {X 0,Y 608.45,Z 242.313,A -85,B 0,C 180,E1 -497.04,E2 -497.04} C_VEL
LIN {X 0,Y 608.446,Z 242.315,A -85,B 0,C 180,E1 -499.696,E2 -499.696} C_VEL
LIN {X 0,Y 608.465,Z 242.321,A -85,B 0,C 180,E1 -502.253,E2 -502.253} C_VEL
LIN {X 0,Y 608.479,Z 242.308,A -85,B 0,C 180,E1 -505.089,E2 -505.089} C_VEL
LIN {X 0,Y 608.458,Z 242.319,A -85,B 0,C 180,E1 -507.905,E2 -507.905} C_VEL
LIN {X 0,Y 608.473,Z 242.317,A -85,B 0,C 180,E1 -510.221,E2 -510.221} C_VEL
LIN {X 0,Y 608.45,Z 242.313,A -85,B 0,C 180,E1 -513.226,E2 -513.226} C_VEL
LIN {X 0,Y 608.47,Z 242.317,A -85,B 0,C 180,E1 -516.155,E2 -516.155} C_VEL
LIN {X 0,Y 608.447,Z 242.313,A -85,B 0,C 180,E1 -519.018,E2 -519.018} C_VEL
LIN {X 0,Y 608.445,Z 242.324,A -85,B 0,C 180,E1 -521.828,E2 -521.828} C_VEL
LIN {X 0,Y 608.471,Z 242.31,A -85,B 0,C 180,E1 -524.594,E2 -524.594} C_VEL
LIN {X 0,Y 608.473,Z 242.314,A -85,B 0,C 180,E1 -527.323,E2 -527.323} C_VEL
LIN {X 0,Y 608.45,Z 242.318,A -85,B 0,C 180,E1 -530.023,E2 -530.023} C_VEL
LIN {X 0,Y 608.477,Z 242.309,A -85,B 0,C 180,E1 -532.701,E2 -532.701} C_VEL
LIN {X 0,Y 608.451,Z 242.319,A -85,B 0,C 180,E1 -535.362,E2 -535.362} C_VEL
LIN {X 0,Y 608.449,Z 242.316,A -85,B 0,C 180,E1 -538.014,E2 -538.014} C_VEL
LIN {X 0,Y 608.476,Z 242.31,A -85,B 0,C 180,E1 -540.662,E2 -540.662} C_VEL
LIN {X 0,Y 608.476,Z 242.317,A -85,B 0,C 180,E1 -543.311,E2 -543.311} C_VEL
LIN {X 0,Y 608.452,Z 242.314,A -85,B 0,C 180,E1 -545.967,E2 -545.967} C_VEL
LIN {X 0,Y 608.455,Z 242.313,A -85,B 0,C 180,E1 -548.636,E2 -548.636} C_VEL
LIN {X 0,Y 608.457,Z 242.319,A -85,B 0,C 180,E1 -549.467,E2 -549.467} C_VEL
LIN {X 0,Y 607.773,Z 242.399,A -85,B 0,C 180,E1 -550.02,E2 -550.02} C_VEL
LIN {X 0,Y 604.915,Z 242.757,A -85,B 0,C 180,E1 -550.917,E2 -550.917} C_VEL
LIN {X 0,Y 602.513,Z 243.057,A -85,B 0,C 180,E1 -551.638,E2 -551.638} C_VEL
LIN {X 0,Y 601.487,Z 243.181,A -85,B 0,C 180,E1 -552.195,E2 -552.195} C_VEL
LIN {X 0,Y 601.405,Z 243.19,A -85,B 0,C 180,E1 -552.383,E2 -552.383} C_VEL
LIN {X 0,Y 601.426,Z 243.192,A -85,B 0,C 180,E1 -554.897,E2 -554.897} C_VEL
LIN {X 0,Y 601.427,Z 243.194,A -85,B 0,C 180,E1 -556.986,E2 -556.986} C_VEL
LIN {X 0,Y 601.405,Z 243.191,A -85,B 0,C 180,E1 -559.81,E2 -559.81} C_VEL
LIN {X 0,Y 601.404,Z 243.194,A -85,B 0,C 180,E1 -562.683,E2 -562.683} C_VEL
LIN {X 0,Y 601.402,Z 243.198,A -85,B 0,C 180,E1 -564.879,E2 -564.879} C_VEL
LIN {X 0,Y 601.417,Z 243.189,A -85,B 0,C 180,E1 -567.868,E2 -567.868} C_VEL
LIN {X 0,Y 601.442,Z 243.186,A -85,B 0,C 180,E1 -570.163,E2 -570.163} C_VEL
LIN {X 0,Y 601.415,Z 243.195,A -85,B 0,C 180,E1 -572.716,E2 -572.716} C_VEL
LIN {X 0,Y 601.412,Z 243.195,A -85,B 0,C 180,E1 -575.116,E2 -575.116} C_VEL
LIN {X 0,Y 601.429,Z 243.189,A -85,B 0,C 180,E1 -577.42,E2 -577.42} C_VEL
LIN {X 0,Y 601.408,Z 243.19,A -85,B 0,C 180,E1 -579.996,E2 -579.996} C_VEL
LIN {X 0,Y 601.406,Z 243.199,A -85,B 0,C 180,E1 -582.671,E2 -582.671} C_VEL
LIN {X 0,Y 601.422,Z 243.189,A -85,B 0,C 180,E1 -585.483,E2 -585.483} C_VEL
LIN {X 0,Y 601.424,Z 243.194,A -85,B 0,C 180,E1 -588.407,E2 -588.407} C_VEL
LIN {X 0,Y 601.409,Z 243.195,A -85,B 0,C 180,E1 -590.874,E2 -590.874} C_VEL
LIN {X 0,Y 601.44,Z 243.187,A -85,B 0,C 180,E1 -593.735,E2 -593.735} C_VEL
LIN {X 0,Y 601.429,Z 243.194,A -85,B 0,C 180,E1 -596.687,E2 -596.687} C_VEL
LIN {X 0,Y 601.41,Z 243.191,A -85,B 0,C 180,E1 -599.058,E2 -599.058} C_VEL
LIN {X 0,Y 601.432,Z 243.186,A -85,B 0,C 180,E1 -601.374,E2 -601.374} C_VEL
LIN {X 0,Y 601.418,Z 243.196,A -85,B 0,C 180,E1 -604.132,E2 -604.132} C_VEL
LIN {X 0,Y 601.417,Z 243.197,A -85,B 0,C 180,E1 -606.59,E2 -606.59} C_VEL
LIN {X 0,Y 601.471,Z 243.338,A -85,B 0,C 180,E1 -608.089,E2 -608.089} C_VEL
LIN {X 0,Y 601.637,Z 251.494,A -85,B 0,C 180,E1 -609.262,E2 -609.262} C_VEL
LIN {X 0,Y 601.533,Z 270.896,A -85,B 0,C 180,E1 -611.965,E2 -611.965} C_VEL
LIN {X 0,Y 601.519,Z 286.324,A -85,B 0,C 180,E1 -614.064,E2 -614.064} C_VEL
LIN {X 0,Y 601.828,Z 289.515,A -85,B 0,C 180,E1 -614.138,E2 -614.138} C_VEL
LIN {X 0,Y 601.731,Z 423.063,A -85,B 0,C 180,E1 -615.767,E2 -615.767} C_VEL
LIN {X 0,Y 601.712,Z 437.51,A -85,B 0,C 180,E1 -616.081,E2 -616.081} C_VEL
LIN {X 0,Y 601.673,Z 450.539,A -85,B 0,C 180,E1 -616.49,E2 -616.49} C_VEL
LIN {X 0,Y 601.632,Z 462.965,A -85,B 0,C 180,E1 -617.005,E2 -617.005} C_VEL
LIN {X 0,Y 601.561,Z 475.945,A -85,B 0,C 180,E1 -617.689,E2 -617.689} C_VEL
LIN {X 0,Y 601.513,Z 487.703,A -85,B 0,C 180,E1 -618.458,E2 -618.458} C_VEL
LIN {X 0,Y 601.481,Z 499.422,A -85,B 0,C 180,E1 -619.396,E2 -619.396} C_VEL
LIN {X 0,Y 601.431,Z 509.905,A -85,B 0,C 180,E1 -620.415,E2 -620.415} C_VEL
LIN {X 0,Y 601.406,Z 518.556,A -85,B 0,C 180,E1 -621.431,E2 -621.431} C_VEL
LIN {X 0,Y 601.391,Z 526.843,A -85,B 0,C 180,E1 -622.614,E2 -622.614} C_VEL
LIN {X 0,Y 601.361,Z 532.512,A -85,B 0,C 180,E1 -623.605,E2 -623.605} C_VEL
LIN {X 0,Y 601.354,Z 537.378,A -85,B 0,C 180,E1 -624.635,E2 -624.635} C_VEL
LIN {X 0,Y 601.345,Z 542.3,A -85,B 0,C 180,E1 -625.979,E2 -625.979} C_VEL
LIN {X 0,Y 601.324,Z 545.735,A -85,B 0,C 180,E1 -627.32,E2 -627.32} C_VEL
LIN {X 0,Y 601.346,Z 547.779,A -85,B 0,C 180,E1 -628.661,E2 -628.661} C_VEL
LIN {X 0,Y 601.334,Z 548.496,A -85,B 0,C 180,E1 -630,E2 -630} C_VEL
LIN {X 0,Y 601.343,Z 547.882,A -85,B 0,C 180,E1 -631.339,E2 -631.339} C_VEL
LIN {X 0,Y 601.321,Z 545.927,A -85,B 0,C 180,E1 -632.679,E2 -632.679} C_VEL
LIN {X 0,Y 601.346,Z 542.584,A -85,B 0,C 180,E1 -634.021,E2 -634.021} C_VEL
LIN {X 0,Y 601.355,Z 537.759,A -85,B 0,C 180,E1 -635.365,E2 -635.365} C_VEL
LIN {X 0,Y 601.368,Z 531.889,A -85,B 0,C 180,E1 -636.601,E2 -636.601} C_VEL
LIN {X 0,Y 601.386,Z 525.219,A -85,B 0,C 180,E1 -637.723,E2 -637.723} C_VEL
LIN {X 0,Y 601.411,Z 516.561,A -85,B 0,C 180,E1 -638.907,E2 -638.907} C_VEL
LIN {X 0,Y 601.432,Z 507.514,A -85,B 0,C 180,E1 -639.925,E2 -639.925} C_VEL
LIN {X 0,Y 601.474,Z 496.336,A -85,B 0,C 180,E1 -640.964,E2 -640.964} C_VEL
LIN {X 0,Y 601.542,Z 484.103,A -85,B 0,C 180,E1 -641.883,E2 -641.883} C_VEL
LIN {X 0,Y 601.561,Z 471.471,A -85,B 0,C 180,E1 -642.653,E2 -642.653} C_VEL
LIN {X 0,Y 601.63,Z 459.198,A -85,B 0,C 180,E1 -643.253,E2 -643.253} C_VEL
LIN {X 0,Y 601.697,Z 445.161,A -85,B 0,C 180,E1 -643.783,E2 -643.783} C_VEL
LIN {X 0,Y 601.729,Z 431.543,A -85,B 0,C 180,E1 -644.155,E2 -644.155} C_VEL
LIN {X 0,Y 601.754,Z 417.595,A -85,B 0,C 180,E1 -644.401,E2 -644.401} C_VEL
LIN {X 0,Y 601.671,Z 287.425,A -85,B 0,C 180,E1 -645.983,E2 -645.983} C_VEL
LIN {X 0,Y 601.503,Z 285.909,A -85,B 0,C 180,E1 -646.067,E2 -646.067} C_VEL
LIN {X 0,Y 601.531,Z 267.303,A -85,B 0,C 180,E1 -648.623,E2 -648.623} C_VEL
LIN {X 0,Y 601.667,Z 246.091,A -85,B 0,C 180,E1 -651.589,E2 -651.589} C_VEL
LIN {X 0,Y 601.436,Z 243.277,A -85,B 0,C 180,E1 -652.047,E2 -652.047} C_VEL
LIN {X 0,Y 601.397,Z 243.192,A -85,B 0,C 180,E1 -654.878,E2 -654.878} C_VEL
LIN {X 0,Y 601.42,Z 243.196,A -85,B 0,C 180,E1 -657.867,E2 -657.867} C_VEL
LIN {X 0,Y 601.427,Z 243.191,A -85,B 0,C 180,E1 -660.163,E2 -660.163} C_VEL
LIN {X 0,Y 601.423,Z 243.188,A -85,B 0,C 180,E1 -662.715,E2 -662.715} C_VEL
LIN {X 0,Y 601.393,Z 243.195,A -85,B 0,C 180,E1 -665.111,E2 -665.111} C_VEL
LIN {X 0,Y 601.431,Z 243.196,A -85,B 0,C 180,E1 -667.418,E2 -667.418} C_VEL
LIN {X 0,Y 601.407,Z 243.193,A -85,B 0,C 180,E1 -669.994,E2 -669.994} C_VEL
LIN {X 0,Y 601.409,Z 243.19,A -85,B 0,C 180,E1 -672.669,E2 -672.669} C_VEL
LIN {X 0,Y 601.421,Z 243.197,A -85,B 0,C 180,E1 -675.481,E2 -675.481} C_VEL
LIN {X 0,Y 601.418,Z 243.188,A -85,B 0,C 180,E1 -678.406,E2 -678.406} C_VEL
LIN {X 0,Y 601.429,Z 243.191,A -85,B 0,C 180,E1 -680.875,E2 -680.875} C_VEL
LIN {X 0,Y 601.439,Z 243.189,A -85,B 0,C 180,E1 -683.733,E2 -683.733} C_VEL
LIN {X 0,Y 601.427,Z 243.186,A -85,B 0,C 180,E1 -686.063,E2 -686.063} C_VEL
LIN {X 0,Y 601.434,Z 243.188,A -85,B 0,C 180,E1 -688.541,E2 -688.541} C_VEL
LIN {X 0,Y 601.429,Z 243.193,A -85,B 0,C 180,E1 -691.373,E2 -691.373} C_VEL
LIN {X 0,Y 601.398,Z 243.193,A -85,B 0,C 180,E1 -693.636,E2 -693.636} C_VEL
LIN {X 0,Y 601.416,Z 243.193,A -85,B 0,C 180,E1 -696.589,E2 -696.589} C_VEL
LIN {X 0,Y 601.426,Z 243.19,A -85,B 0,C 180,E1 -699.478,E2 -699.478} C_VEL
LIN {X 0,Y 601.394,Z 243.194,A -85,B 0,C 180,E1 -702.311,E2 -702.311} C_VEL
LIN {X 0,Y 601.414,Z 243.193,A -85,B 0,C 180,E1 -704.409,E2 -704.409} C_VEL
LIN {X 0,Y 601.422,Z 243.192,A -85,B 0,C 180,E1 -707.172,E2 -707.172} C_VEL
LIN {X 0,Y 601.426,Z 243.188,A -85,B 0,C 180,E1 -709.905,E2 -709.905} C_VEL
LIN {X 0,Y 601.446,Z 243.194,A -85,B 0,C 180,E1 -712.615,E2 -712.615} C_VEL
LIN {X 0,Y 601.423,Z 243.189,A -85,B 0,C 180,E1 -715.308,E2 -715.308} C_VEL
LIN {X 0,Y 601.417,Z 243.19,A -85,B 0,C 180,E1 -717.991,E2 -717.991} C_VEL
LIN {X 0,Y 601.449,Z 243.193,A -85,B 0,C 180,E1 -720.669,E2 -720.669} C_VEL
LIN {X 0,Y 601.427,Z 243.187,A -85,B 0,C 180,E1 -723.35,E2 -723.35} C_VEL
LIN {X 0,Y 601.405,Z 243.194,A -85,B 0,C 180,E1 -726.037,E2 -726.037} C_VEL
LIN {X 0,Y 601.434,Z 243.191,A -85,B 0,C 180,E1 -728.738,E2 -728.738} C_VEL
LIN {X 0,Y 601.428,Z 243.187,A -85,B 0,C 180,E1 -731.458,E2 -731.458} C_VEL
LIN {X 0,Y 601.41,Z 243.199,A -85,B 0,C 180,E1 -734.206,E2 -734.206} C_VEL
LIN {X 0,Y 601.427,Z 243.188,A -85,B 0,C 180,E1 -736.986,E2 -736.986} C_VEL
LIN {X 0,Y 601.406,Z 243.195,A -85,B 0,C 180,E1 -739.809,E2 -739.809} C_VEL
LIN {X 0,Y 601.403,Z 243.192,A -85,B 0,C 180,E1 -742.683,E2 -742.683} C_VEL
LIN {X 0,Y 601.4,Z 243.191,A -85,B 0,C 180,E1 -744.879,E2 -744.879} C_VEL
LIN {X 0,Y 601.416,Z 243.197,A -85,B 0,C 180,E1 -747.868,E2 -747.868} C_VEL
LIN {X 0,Y 601.441,Z 243.193,A -85,B 0,C 180,E1 -750.163,E2 -750.163} C_VEL
LIN {X 0,Y 601.412,Z 243.189,A -85,B 0,C 180,E1 -752.716,E2 -752.716} C_VEL
LIN {X 0,Y 601.411,Z 243.189,A -85,B 0,C 180,E1 -755.116,E2 -755.116} C_VEL
LIN {X 0,Y 601.429,Z 243.191,A -85,B 0,C 180,E1 -757.42,E2 -757.42} C_VEL
LIN {X 0,Y 601.406,Z 243.197,A -85,B 0,C 180,E1 -759.996,E2 -759.996} C_VEL
LIN {X 0,Y 601.406,Z 243.19,A -85,B 0,C 180,E1 -762.671,E2 -762.671} C_VEL
LIN {X 0,Y 601.421,Z 243.196,A -85,B 0,C 180,E1 -765.483,E2 -765.483} C_VEL
LIN {X 0,Y 601.422,Z 243.188,A -85,B 0,C 180,E1 -768.407,E2 -768.407} C_VEL
LIN {X 0,Y 601.43,Z 243.188,A -85,B 0,C 180,E1 -770.876,E2 -770.876} C_VEL
LIN {X 0,Y 601.398,Z 243.2,A -85,B 0,C 180,E1 -773.418,E2 -773.418} C_VEL
LIN {X 0,Y 601.431,Z 243.189,A -85,B 0,C 180,E1 -776.065,E2 -776.065} C_VEL
LIN {X 0,Y 601.439,Z 243.186,A -85,B 0,C 180,E1 -778.543,E2 -778.543} C_VEL
LIN {X 0,Y 601.432,Z 243.197,A -85,B 0,C 180,E1 -781.374,E2 -781.374} C_VEL
LIN {X 0,Y 601.4,Z 243.197,A -85,B 0,C 180,E1 -783.637,E2 -783.637} C_VEL
LIN {X 0,Y 601.419,Z 243.193,A -85,B 0,C 180,E1 -786.59,E2 -786.59} C_VEL
LIN {X 0,Y 601.469,Z 243.431,A -85,B 0,C 180,E1 -787.07,E2 -787.07} C_VEL
LIN {X 0,Y 601.697,Z 247.842,A -85,B 0,C 180,E1 -787.694,E2 -787.694} C_VEL
LIN {X 0,Y 601.559,Z 270.644,A -85,B 0,C 180,E1 -790.729,E2 -790.729} C_VEL
LIN {X 0,Y 601.472,Z 289.867,A -85,B 0,C 180,E1 -793.246,E2 -793.246} C_VEL
LIN {X 0,Y 601.564,Z 296.212,A -85,B 0,C 180,E1 -794.033,E2 -794.033} C_VEL
LIN {X 0,Y 601.835,Z 299.648,A -85,B 0,C 180,E1 -794.094,E2 -794.094} C_VEL
LIN {X 0,Y 601.755,Z 432.93,A -85,B 0,C 180,E1 -795.721,E2 -795.721} C_VEL
LIN {X 0,Y 601.715,Z 447.274,A -85,B 0,C 180,E1 -796.029,E2 -796.029} C_VEL
LIN {X 0,Y 601.659,Z 459.926,A -85,B 0,C 180,E1 -796.422,E2 -796.422} C_VEL
LIN {X 0,Y 601.628,Z 472.101,A -85,B 0,C 180,E1 -796.919,E2 -796.919} C_VEL
LIN {X 0,Y 601.551,Z 485.27,A -85,B 0,C 180,E1 -797.604,E2 -797.604} C_VEL
LIN {X 0,Y 601.511,Z 497.154,A -85,B 0,C 180,E1 -798.373,E2 -798.373} C_VEL
LIN {X 0,Y 601.49,Z 507.996,A -85,B 0,C 180,E1 -799.225,E2 -799.225} C_VEL
LIN {X 0,Y 601.422,Z 518.71,A -85,B 0,C 180,E1 -800.245,E2 -800.245} C_VEL
LIN {X 0,Y 601.407,Z 527.56,A -85,B 0,C 180,E1 -801.262,E2 -801.262} C_VEL
LIN {X 0,Y 601.406,Z 536.041,A -85,B 0,C 180,E1 -802.446,E2 -802.446} C_VEL
LIN {X 0,Y 601.361,Z 542.751,A -85,B 0,C 180,E1 -803.604,E2 -803.604} C_VEL
LIN {X 0,Y 601.355,Z 547.568,A -85,B 0,C 180,E1 -804.635,E2 -804.635} C_VEL
LIN {X 0,Y 601.343,Z 552.442,A -85,B 0,C 180,E1 -805.979,E2 -805.979} C_VEL
LIN {X 0,Y 601.324,Z 555.831,A -85,B 0,C 180,E1 -807.321,E2 -807.321} C_VEL
LIN {X 0,Y 601.342,Z 557.831,A -85,B 0,C 180,E1 -808.661,E2 -808.661} C_VEL
LIN {X 0,Y 601.333,Z 558.5,A -85,B 0,C 180,E1 -810,E2 -810} C_VEL
LIN {X 0,Y 601.342,Z 557.831,A -85,B 0,C 180,E1 -811.339,E2 -811.339} C_VEL
LIN {X 0,Y 601.324,Z 555.832,A -85,B 0,C 180,E1 -812.68,E2 -812.68} C_VEL
LIN {X 0,Y 601.343,Z 552.442,A -85,B 0,C 180,E1 -814.021,E2 -814.021} C_VEL
LIN {X 0,Y 601.355,Z 547.568,A -85,B 0,C 180,E1 -815.365,E2 -815.365} C_VEL
LIN {X 0,Y 601.372,Z 541.623,A -85,B 0,C 180,E1 -816.605,E2 -816.605} C_VEL
LIN {X 0,Y 601.386,Z 534.92,A -85,B 0,C 180,E1 -817.723,E2 -817.723} C_VEL
LIN {X 0,Y 601.412,Z 526.199,A -85,B 0,C 180,E1 -818.907,E2 -818.907} C_VEL
LIN {X 0,Y 601.433,Z 517.083,A -85,B 0,C 180,E1 -819.925,E2 -819.925} C_VEL
LIN {X 0,Y 601.497,Z 506.828,A -85,B 0,C 180,E1 -820.877,E2 -820.877} C_VEL
LIN {X 0,Y 601.533,Z 495.973,A -85,B 0,C 180,E1 -821.712,E2 -821.712} C_VEL
LIN {X 0,Y 601.574,Z 483.781,A -85,B 0,C 180,E1 -822.482,E2 -822.482} C_VEL
LIN {X 0,Y 601.628,Z 472.099,A -85,B 0,C 180,E1 -823.081,E2 -823.081} C_VEL
LIN {X 0,Y 601.669,Z 458.945,A -85,B 0,C 180,E1 -823.612,E2 -823.612} C_VEL
LIN {X 0,Y 601.706,Z 445.035,A -85,B 0,C 180,E1 -824.028,E2 -824.028} C_VEL
LIN {X 0,Y 601.732,Z 430.561,A -85,B 0,C 180,E1 -824.314,E2 -824.314} C_VEL
LIN {X 0,Y 601.729,Z 297.205,A -85,B 0,C 180,E1 -825.938,E2 -825.938} C_VEL
LIN {X 0,Y 601.512,Z 295.525,A -85,B 0,C 180,E1 -826.023,E2 -826.023} C_VEL
LIN {X 0,Y 601.518,Z 274.733,A -85,B 0,C 180,E1 -828.733,E2 -828.733} C_VEL
LIN {X 0,Y 601.612,Z 257.777,A -85,B 0,C 180,E1 -830.977,E2 -830.977} C_VEL
LIN {X 0,Y 601.704,Z 245.131,A -85,B 0,C 180,E1 -832.671,E2 -832.671} C_VEL
LIN {X 0,Y 601.463,Z 243.343,A -85,B 0,C 180,E1 -832.953,E2 -832.953} C_VEL
LIN {X 0,Y 601.436,Z 243.187,A -85,B 0,C 180,E1 -835.617,E2 -835.617} C_VEL
LIN {X 0,Y 601.4,Z 243.192,A -85,B 0,C 180,E1 -837.868,E2 -837.868} C_VEL
LIN {X 0,Y 601.425,Z 243.19,A -85,B 0,C 180,E1 -840.163,E2 -840.163} C_VEL
LIN {X 0,Y 601.421,Z 243.196,A -85,B 0,C 180,E1 -842.715,E2 -842.715} C_VEL
LIN {X 0,Y 601.396,Z 243.193,A -85,B 0,C 180,E1 -845.112,E2 -845.112} C_VEL
LIN {X 0,Y 601.431,Z 243.187,A -85,B 0,C 180,E1 -847.418,E2 -847.418} C_VEL
LIN {X 0,Y 601.398,Z 243.195,A -85,B 0,C 180,E1 -849.995,E2 -849.995} C_VEL
LIN {X 0,Y 601.412,Z 243.195,A -85,B 0,C 180,E1 -852.669,E2 -852.669} C_VEL
LIN {X 0,Y 601.421,Z 243.189,A -85,B 0,C 180,E1 -855.481,E2 -855.481} C_VEL
LIN {X 0,Y 601.42,Z 243.196,A -85,B 0,C 180,E1 -858.406,E2 -858.406} C_VEL
LIN {X 0,Y 601.434,Z 243.188,A -85,B 0,C 180,E1 -860.875,E2 -860.875} C_VEL
LIN {X 0,Y 601.439,Z 243.189,A -85,B 0,C 180,E1 -863.733,E2 -863.733} C_VEL
LIN {X 0,Y 601.428,Z 243.196,A -85,B 0,C 180,E1 -866.063,E2 -866.063} C_VEL
LIN {X 0,Y 601.426,Z 243.188,A -85,B 0,C 180,E1 -869.058,E2 -869.058} C_VEL
LIN {X 0,Y 601.424,Z 243.189,A -85,B 0,C 180,E1 -871.373,E2 -871.373} C_VEL
LIN {X 0,Y 601.4,Z 243.195,A -85,B 0,C 180,E1 -873.636,E2 -873.636} C_VEL
LIN {X 0,Y 601.417,Z 243.19,A -85,B 0,C 180,E1 -876.59,E2 -876.59} C_VEL
LIN {X 0,Y 601.424,Z 243.192,A -85,B 0,C 180,E1 -879.478,E2 -879.478} C_VEL
LIN {X 0,Y 601.397,Z 243.194,A -85,B 0,C 180,E1 -882.312,E2 -882.312} C_VEL
LIN {X 0,Y 601.414,Z 243.191,A -85,B 0,C 180,E1 -884.409,E2 -884.409} C_VEL
LIN {X 0,Y 601.42,Z 243.191,A -85,B 0,C 180,E1 -887.172,E2 -887.172} C_VEL
LIN {X 0,Y 601.427,Z 243.194,A -85,B 0,C 180,E1 -889.905,E2 -889.905} C_VEL
LIN {X 0,Y 601.446,Z 243.185,A -85,B 0,C 180,E1 -892.615,E2 -892.615} C_VEL
LIN {X 0,Y 601.419,Z 243.194,A -85,B 0,C 180,E1 -895.308,E2 -895.308} C_VEL
LIN {X 0,Y 601.419,Z 243.192,A -85,B 0,C 180,E1 -897.991,E2 -897.991} C_VEL
LIN {X 0,Y 601.446,Z 243.185,A -85,B 0,C 180,E1 -900.67,E2 -900.67} C_VEL
LIN {X 0,Y 601.427,Z 243.196,A -85,B 0,C 180,E1 -903.35,E2 -903.35} C_VEL
LIN {X 0,Y 601.405,Z 243.192,A -85,B 0,C 180,E1 -906.037,E2 -906.037} C_VEL
LIN {X 0,Y 601.434,Z 243.188,A -85,B 0,C 180,E1 -908.738,E2 -908.738} C_VEL
LIN {X 0,Y 601.428,Z 243.195,A -85,B 0,C 180,E1 -911.458,E2 -911.458} C_VEL
LIN {X 0,Y 601.405,Z 243.19,A -85,B 0,C 180,E1 -912.383,E2 -912.383} C_VEL
LIN {X 0,Y 600.744,Z 243.279,A -85,B 0,C 180,E1 -912.943,E2 -912.943} C_VEL
LIN {X 0,Y 597.894,Z 243.635,A -85,B 0,C 180,E1 -913.85,E2 -913.85} C_VEL
LIN {X 0,Y 595.482,Z 243.936,A -85,B 0,C 180,E1 -914.581,E2 -914.581} C_VEL
LIN {X 0,Y 594.443,Z 244.066,A -85,B 0,C 180,E1 -915.144,E2 -915.144} C_VEL
LIN {X 0,Y 594.358,Z 244.072,A -85,B 0,C 180,E1 -915.335,E2 -915.335} C_VEL
LIN {X 0,Y 594.374,Z 244.067,A -85,B 0,C 180,E1 -917.904,E2 -917.904} C_VEL
LIN {X 0,Y 594.372,Z 244.073,A -85,B 0,C 180,E1 -920.918,E2 -920.918} C_VEL
LIN {X 0,Y 594.387,Z 244.066,A -85,B 0,C 180,E1 -923.704,E2 -923.704} C_VEL
LIN {X 0,Y 594.383,Z 244.069,A -85,B 0,C 180,E1 -926.7,E2 -926.7} C_VEL
LIN {X 0,Y 594.375,Z 244.076,A -85,B 0,C 180,E1 -928.999,E2 -928.999} C_VEL
LIN {X 0,Y 594.386,Z 244.064,A -85,B 0,C 180,E1 -931.646,E2 -931.646} C_VEL
LIN {X 0,Y 594.394,Z 244.067,A -85,B 0,C 180,E1 -934.579,E2 -934.579} C_VEL
LIN {X 0,Y 594.381,Z 244.072,A -85,B 0,C 180,E1 -937.087,E2 -937.087} C_VEL
LIN {X 0,Y 594.372,Z 244.066,A -85,B 0,C 180,E1 -939.775,E2 -939.775} C_VEL
LIN {X 0,Y 594.364,Z 244.07,A -85,B 0,C 180,E1 -942.376,E2 -942.376} C_VEL
LIN {X 0,Y 594.36,Z 244.071,A -85,B 0,C 180,E1 -945.192,E2 -945.192} C_VEL
LIN {X 0,Y 594.369,Z 244.065,A -85,B 0,C 180,E1 -947.626,E2 -947.626} C_VEL
LIN {X 0,Y 594.387,Z 244.071,A -85,B 0,C 180,E1 -950.321,E2 -950.321} C_VEL
LIN {X 0,Y 594.382,Z 244.07,A -85,B 0,C 180,E1 -952.914,E2 -952.914} C_VEL
LIN {X 0,Y 594.381,Z 244.067,A -85,B 0,C 180,E1 -955.862,E2 -955.862} C_VEL
LIN {X 0,Y 594.369,Z 244.074,A -85,B 0,C 180,E1 -958.65,E2 -958.65} C_VEL
LIN {X 0,Y 594.383,Z 244.066,A -85,B 0,C 180,E1 -961.043,E2 -961.043} C_VEL
LIN {X 0,Y 594.391,Z 244.069,A -85,B 0,C 180,E1 -963.977,E2 -963.977} C_VEL
LIN {X 0,Y 594.388,Z 244.075,A -85,B 0,C 180,E1 -966.296,E2 -966.296} C_VEL
LIN {X 0,Y 594.433,Z 244.274,A -85,B 0,C 180,E1 -967.953,E2 -967.953} C_VEL
LIN {X 0,Y 594.72,Z 249.064,A -85,B 0,C 180,E1 -968.662,E2 -968.662} C_VEL
LIN {X 0,Y 594.563,Z 269.628,A -85,B 0,C 180,E1 -971.567,E2 -971.567} C_VEL
LIN {X 0,Y 594.533,Z 286.326,A -85,B 0,C 180,E1 -973.872,E2 -973.872} C_VEL
LIN {X 0,Y 595.016,Z 289.561,A -85,B 0,C 180,E1 -973.951,E2 -973.951} C_VEL
LIN {X 0,Y 594.851,Z 423.83,A -85,B 0,C 180,E1 -975.613,E2 -975.613} C_VEL
LIN {X 0,Y 594.805,Z 438.286,A -85,B 0,C 180,E1 -975.937,E2 -975.937} C_VEL
LIN {X 0,Y 594.754,Z 452.802,A -85,B 0,C 180,E1 -976.417,E2 -976.417} C_VEL
LIN {X 0,Y 594.644,Z 466.485,A -85,B 0,C 180,E1 -977.023,E2 -977.023} C_VEL
LIN {X 0,Y 594.563,Z 478.779,A -85,B 0,C 180,E1 -977.716,E2 -977.716} C_VEL
LIN {X 0,Y 594.528,Z 491.048,A -85,B 0,C 180,E1 -978.569,E2 -978.569} C_VEL
LIN {X 0,Y 594.448,Z 501.362,A -85,B 0,C 180,E1 -979.441,E2 -979.441} C_VEL
LIN {X 0,Y 594.371,Z 511.462,A -85,B 0,C 180,E1 -980.472,E2 -980.472} C_VEL
LIN {X 0,Y 594.324,Z 519.846,A -85,B 0,C 180,E1 -981.5,E2 -981.5} C_VEL
LIN {X 0,Y 594.303,Z 527.86,A -85,B 0,C 180,E1 -982.697,E2 -982.697} C_VEL
LIN {X 0,Y 594.281,Z 534.314,A -85,B 0,C 180,E1 -983.89,E2 -983.89} C_VEL
LIN {X 0,Y 594.235,Z 540.036,A -85,B 0,C 180,E1 -985.251,E2 -985.251} C_VEL
LIN {X 0,Y 594.259,Z 544.199,A -85,B 0,C 180,E1 -986.61,E2 -986.61} C_VEL
LIN {X 0,Y 594.242,Z 546.927,A -85,B 0,C 180,E1 -987.967,E2 -987.967} C_VEL
LIN {X 0,Y 594.235,Z 548.302,A -85,B 0,C 180,E1 -989.322,E2 -989.322} C_VEL
LIN {X 0,Y 594.236,Z 548.356,A -85,B 0,C 180,E1 -990.678,E2 -990.678} C_VEL
LIN {X 0,Y 594.241,Z 547.073,A -85,B 0,C 180,E1 -992.033,E2 -992.033} C_VEL
LIN {X 0,Y 594.259,Z 544.433,A -85,B 0,C 180,E1 -993.39,E2 -993.39} C_VEL
LIN {X 0,Y 594.236,Z 540.363,A -85,B 0,C 180,E1 -994.749,E2 -994.749} C_VEL
LIN {X 0,Y 594.282,Z 534.741,A -85,B 0,C 180,E1 -996.11,E2 -996.11} C_VEL
LIN {X 0,Y 594.303,Z 528.393,A -85,B 0,C 180,E1 -997.303,E2 -997.303} C_VEL
LIN {X 0,Y 594.324,Z 520.497,A -85,B 0,C 180,E1 -998.5,E2 -998.5} C_VEL
LIN {X 0,Y 594.355,Z 512.242,A -85,B 0,C 180,E1 -999.529,E2 -999.529} C_VEL
LIN {X 0,Y 594.449,Z 502.304,A -85,B 0,C 180,E1 -1000.559,E2 -1000.559} C_VEL
LIN {X 0,Y 594.493,Z 491.167,A -85,B 0,C 180,E1 -1001.512,E2 -1001.512} C_VEL
LIN {X 0,Y 594.581,Z 478.834,A -85,B 0,C 180,E1 -1002.371,E2 -1002.371} C_VEL
LIN {X 0,Y 594.665,Z 466.549,A -85,B 0,C 180,E1 -1003.063,E2 -1003.063} C_VEL
LIN {X 0,Y 594.728,Z 452.882,A -85,B 0,C 180,E1 -1003.67,E2 -1003.67} C_VEL
LIN {X 0,Y 594.806,Z 438.47,A -85,B 0,C 180,E1 -1004.147,E2 -1004.147} C_VEL
LIN {X 0,Y 594.871,Z 425.113,A -85,B 0,C 180,E1 -1004.452,E2 -1004.452} C_VEL
LIN {X 0,Y 594.913,Z 398.858,A -85,B 0,C 180,E1 -1004.801,E2 -1004.801} C_VEL
LIN {X 0,Y 594.874,Z 288.496,A -85,B 0,C 180,E1 -1006.156,E2 -1006.156} C_VEL
LIN {X 0,Y 594.535,Z 286.354,A -85,B 0,C 180,E1 -1006.216,E2 -1006.216} C_VEL
LIN {X 0,Y 594.553,Z 268.998,A -85,B 0,C 180,E1 -1008.611,E2 -1008.611} C_VEL
LIN {X 0,Y 594.724,Z 248.632,A -85,B 0,C 180,E1 -1011.489,E2 -1011.489} C_VEL
LIN {X 0,Y 594.416,Z 244.302,A -85,B 0,C 180,E1 -1012.139,E2 -1012.139} C_VEL
LIN {X 0,Y 594.389,Z 244.066,A -85,B 0,C 180,E1 -1014.445,E2 -1014.445} C_VEL
LIN {X 0,Y 594.38,Z 244.066,A -85,B 0,C 180,E1 -1016.699,E2 -1016.699} C_VEL
LIN {X 0,Y 594.381,Z 244.066,A -85,B 0,C 180,E1 -1018.998,E2 -1018.998} C_VEL
LIN {X 0,Y 594.377,Z 244.076,A -85,B 0,C 180,E1 -1021.642,E2 -1021.642} C_VEL
LIN {X 0,Y 594.376,Z 244.066,A -85,B 0,C 180,E1 -1024.579,E2 -1024.579} C_VEL
LIN {X 0,Y 594.38,Z 244.069,A -85,B 0,C 180,E1 -1027.086,E2 -1027.086} C_VEL
LIN {X 0,Y 594.37,Z 244.072,A -85,B 0,C 180,E1 -1029.773,E2 -1029.773} C_VEL
LIN {X 0,Y 594.368,Z 244.066,A -85,B 0,C 180,E1 -1032.374,E2 -1032.374} C_VEL
LIN {X 0,Y 594.359,Z 244.075,A -85,B 0,C 180,E1 -1035.19,E2 -1035.19} C_VEL
LIN {X 0,Y 594.378,Z 244.064,A -85,B 0,C 180,E1 -1038.151,E2 -1038.151} C_VEL
LIN {X 0,Y 594.382,Z 244.074,A -85,B 0,C 180,E1 -1041.195,E2 -1041.195} C_VEL
LIN {X 0,Y 594.391,Z 244.066,A -85,B 0,C 180,E1 -1043.758,E2 -1043.758} C_VEL
LIN {X 0,Y 594.373,Z 244.064,A -85,B 0,C 180,E1 -1046.238,E2 -1046.238} C_VEL
LIN {X 0,Y 594.384,Z 244.067,A -85,B 0,C 180,E1 -1048.65,E2 -1048.65} C_VEL
LIN {X 0,Y 594.378,Z 244.076,A -85,B 0,C 180,E1 -1051.041,E2 -1051.041} C_VEL
LIN {X 0,Y 594.378,Z 244.065,A -85,B 0,C 180,E1 -1053.976,E2 -1053.976} C_VEL
LIN {X 0,Y 594.388,Z 244.066,A -85,B 0,C 180,E1 -1056.296,E2 -1056.296} C_VEL
LIN {X 0,Y 594.397,Z 244.068,A -85,B 0,C 180,E1 -1059.224,E2 -1059.224} C_VEL
LIN {X 0,Y 594.374,Z 244.067,A -85,B 0,C 180,E1 -1062.096,E2 -1062.096} C_VEL
LIN {X 0,Y 594.366,Z 244.068,A -85,B 0,C 180,E1 -1064.219,E2 -1064.219} C_VEL
LIN {X 0,Y 594.369,Z 244.073,A -85,B 0,C 180,E1 -1067.017,E2 -1067.017} C_VEL
LIN {X 0,Y 594.386,Z 244.064,A -85,B 0,C 180,E1 -1069.784,E2 -1069.784} C_VEL
LIN {X 0,Y 594.394,Z 244.071,A -85,B 0,C 180,E1 -1072.527,E2 -1072.527} C_VEL
LIN {X 0,Y 594.392,Z 244.065,A -85,B 0,C 180,E1 -1075.252,E2 -1075.252} C_VEL
LIN {X 0,Y 594.387,Z 244.065,A -85,B 0,C 180,E1 -1077.967,E2 -1077.967} C_VEL
LIN {X 0,Y 594.419,Z 244.068,A -85,B 0,C 180,E1 -1080.677,E2 -1080.677} C_VEL
LIN {X 0,Y 594.378,Z 244.065,A -85,B 0,C 180,E1 -1083.389,E2 -1083.389} C_VEL
LIN {X 0,Y 594.361,Z 244.073,A -85,B 0,C 180,E1 -1086.109,E2 -1086.109} C_VEL
LIN {X 0,Y 594.395,Z 244.066,A -85,B 0,C 180,E1 -1088.842,E2 -1088.842} C_VEL
LIN {X 0,Y 594.386,Z 244.065,A -85,B 0,C 180,E1 -1091.596,E2 -1091.596} C_VEL
LIN {X 0,Y 594.381,Z 244.074,A -85,B 0,C 180,E1 -1094.377,E2 -1094.377} C_VEL
LIN {X 0,Y 594.385,Z 244.064,A -85,B 0,C 180,E1 -1097.193,E2 -1097.193} C_VEL
LIN {X 0,Y 594.372,Z 244.075,A -85,B 0,C 180,E1 -1100.054,E2 -1100.054} C_VEL
LIN {X 0,Y 594.357,Z 244.068,A -85,B 0,C 180,E1 -1102.968,E2 -1102.968} C_VEL
LIN {X 0,Y 594.371,Z 244.067,A -85,B 0,C 180,E1 -1105.193,E2 -1105.193} C_VEL
LIN {X 0,Y 594.376,Z 244.068,A -85,B 0,C 180,E1 -1107.527,E2 -1107.527} C_VEL
LIN {X 0,Y 594.393,Z 244.068,A -85,B 0,C 180,E1 -1110.331,E2 -1110.331} C_VEL
LIN {X 0,Y 594.371,Z 244.065,A -85,B 0,C 180,E1 -1112.951,E2 -1112.951} C_VEL
LIN {X 0,Y 594.378,Z 244.067,A -85,B 0,C 180,E1 -1115.407,E2 -1115.407} C_VEL
LIN {X 0,Y 594.381,Z 244.074,A -85,B 0,C 180,E1 -1117.941,E2 -1117.941} C_VEL
LIN {X 0,Y 594.374,Z 244.066,A -85,B 0,C 180,E1 -1120.823,E2 -1120.823} C_VEL
LIN {X 0,Y 594.361,Z 244.072,A -85,B 0,C 180,E1 -1123.3,E2 -1123.3} C_VEL
LIN {X 0,Y 594.378,Z 244.068,A -85,B 0,C 180,E1 -1126.16,E2 -1126.16} C_VEL
LIN {X 0,Y 594.379,Z 244.064,A -85,B 0,C 180,E1 -1128.537,E2 -1128.537} C_VEL
LIN {X 0,Y 594.382,Z 244.071,A -85,B 0,C 180,E1 -1131.296,E2 -1131.296} C_VEL
LIN {X 0,Y 594.348,Z 244.076,A -85,B 0,C 180,E1 -1133.756,E2 -1133.756} C_VEL
LIN {X 0,Y 594.378,Z 244.066,A -85,B 0,C 180,E1 -1136.24,E2 -1136.24} C_VEL
LIN {X 0,Y 594.388,Z 244.065,A -85,B 0,C 180,E1 -1138.652,E2 -1138.652} C_VEL
LIN {X 0,Y 594.383,Z 244.068,A -85,B 0,C 180,E1 -1141.043,E2 -1141.043} C_VEL
LIN {X 0,Y 594.386,Z 244.067,A -85,B 0,C 180,E1 -1143.978,E2 -1143.978} C_VEL
LIN {X 0,Y 594.388,Z 244.072,A -85,B 0,C 180,E1 -1146.666,E2 -1146.666} C_VEL
LIN {X 0,Y 594.408,Z 244.287,A -85,B 0,C 180,E1 -1146.897,E2 -1146.897} C_VEL
LIN {X 0,Y 594.825,Z 248.252,A -85,B 0,C 180,E1 -1147.478,E2 -1147.478} C_VEL
LIN {X 0,Y 594.652,Z 270.644,A -85,B 0,C 180,E1 -1150.496,E2 -1150.496} C_VEL
LIN {X 0,Y 594.492,Z 289.158,A -85,B 0,C 180,E1 -1152.95,E2 -1152.95} C_VEL
LIN {X 0,Y 594.589,Z 296.203,A -85,B 0,C 180,E1 -1153.84,E2 -1153.84} C_VEL
LIN {X 0,Y 595.032,Z 299.648,A -85,B 0,C 180,E1 -1153.908,E2 -1153.908} C_VEL
LIN {X 0,Y 594.857,Z 433.904,A -85,B 0,C 180,E1 -1155.569,E2 -1155.569} C_VEL
LIN {X 0,Y 594.818,Z 448.156,A -85,B 0,C 180,E1 -1155.889,E2 -1155.889} C_VEL
LIN {X 0,Y 594.729,Z 461.723,A -85,B 0,C 180,E1 -1156.33,E2 -1156.33} C_VEL
LIN {X 0,Y 594.653,Z 475.643,A -85,B 0,C 180,E1 -1156.937,E2 -1156.937} C_VEL
LIN {X 0,Y 594.581,Z 488.101,A -85,B 0,C 180,E1 -1157.629,E2 -1157.629} C_VEL
LIN {X 0,Y 594.524,Z 500.563,A -85,B 0,C 180,E1 -1158.488,E2 -1158.488} C_VEL
LIN {X 0,Y 594.449,Z 511.839,A -85,B 0,C 180,E1 -1159.441,E2 -1159.441} C_VEL
LIN {X 0,Y 594.368,Z 521.852,A -85,B 0,C 180,E1 -1160.472,E2 -1160.472} C_VEL
LIN {X 0,Y 594.324,Z 530.172,A -85,B 0,C 180,E1 -1161.5,E2 -1161.5} C_VEL
LIN {X 0,Y 594.303,Z 538.127,A -85,B 0,C 180,E1 -1162.697,E2 -1162.697} C_VEL
LIN {X 0,Y 594.281,Z 544.528,A -85,B 0,C 180,E1 -1163.89,E2 -1163.89} C_VEL
LIN {X 0,Y 594.237,Z 550.199,A -85,B 0,C 180,E1 -1165.251,E2 -1165.251} C_VEL
LIN {X 0,Y 594.259,Z 554.315,A -85,B 0,C 180,E1 -1166.61,E2 -1166.61} C_VEL
LIN {X 0,Y 594.241,Z 557,A -85,B 0,C 180,E1 -1167.967,E2 -1167.967} C_VEL
LIN {X 0,Y 594.237,Z 558.332,A -85,B 0,C 180,E1 -1169.322,E2 -1169.322} C_VEL
LIN {X 0,Y 594.237,Z 558.332,A -85,B 0,C 180,E1 -1170.678,E2 -1170.678} C_VEL
LIN {X 0,Y 594.242,Z 557,A -85,B 0,C 180,E1 -1172.033,E2 -1172.033} C_VEL
LIN {X 0,Y 594.259,Z 554.316,A -85,B 0,C 180,E1 -1173.39,E2 -1173.39} C_VEL
LIN {X 0,Y 594.237,Z 550.199,A -85,B 0,C 180,E1 -1174.749,E2 -1174.749} C_VEL
LIN {X 0,Y 594.281,Z 544.527,A -85,B 0,C 180,E1 -1176.11,E2 -1176.11} C_VEL
LIN {X 0,Y 594.303,Z 538.126,A -85,B 0,C 180,E1 -1177.303,E2 -1177.303} C_VEL
LIN {X 0,Y 594.324,Z 530.171,A -85,B 0,C 180,E1 -1178.5,E2 -1178.5} C_VEL
LIN {X 0,Y 594.367,Z 521.852,A -85,B 0,C 180,E1 -1179.528,E2 -1179.528} C_VEL
LIN {X 0,Y 594.449,Z 511.838,A -85,B 0,C 180,E1 -1180.559,E2 -1180.559} C_VEL
LIN {X 0,Y 594.523,Z 500.564,A -85,B 0,C 180,E1 -1181.512,E2 -1181.512} C_VEL
LIN {X 0,Y 594.58,Z 488.1,A -85,B 0,C 180,E1 -1182.371,E2 -1182.371} C_VEL
LIN {X 0,Y 594.653,Z 475.642,A -85,B 0,C 180,E1 -1183.063,E2 -1183.063} C_VEL
LIN {X 0,Y 594.743,Z 461.718,A -85,B 0,C 180,E1 -1183.67,E2 -1183.67} C_VEL
LIN {X 0,Y 594.819,Z 448.137,A -85,B 0,C 180,E1 -1184.111,E2 -1184.111} C_VEL
LIN {X 0,Y 594.874,Z 433.898,A -85,B 0,C 180,E1 -1184.43,E2 -1184.43} C_VEL
LIN {X 0,Y 594.856,Z 297.852,A -85,B 0,C 180,E1 -1186.119,E2 -1186.119} C_VEL
LIN {X 0,Y 594.541,Z 295.718,A -85,B 0,C 180,E1 -1186.194,E2 -1186.194} C_VEL
LIN {X 0,Y 594.569,Z 275.435,A -85,B 0,C 180,E1 -1188.867,E2 -1188.867} C_VEL
LIN {X 0,Y 594.699,Z 258.156,A -85,B 0,C 180,E1 -1191.181,E2 -1191.181} C_VEL
LIN {X 0,Y 594.742,Z 246.081,A -85,B 0,C 180,E1 -1192.821,E2 -1192.821} C_VEL
LIN {X 0,Y 594.387,Z 244.163,A -85,B 0,C 180,E1 -1193.15,E2 -1193.15} C_VEL
LIN {X 0,Y 594.373,Z 244.068,A -85,B 0,C 180,E1 -1195.944,E2 -1195.944} C_VEL
LIN {X 0,Y 594.375,Z 244.071,A -85,B 0,C 180,E1 -1198.226,E2 -1198.226} C_VEL
LIN {X 0,Y 594.381,Z 244.073,A -85,B 0,C 180,E1 -1200.559,E2 -1200.559} C_VEL
LIN {X 0,Y 594.377,Z 244.069,A -85,B 0,C 180,E1 -1202.949,E2 -1202.949} C_VEL
LIN {X 0,Y 594.349,Z 244.07,A -85,B 0,C 180,E1 -1205.408,E2 -1205.408} C_VEL
LIN {X 0,Y 594.381,Z 244.067,A -85,B 0,C 180,E1 -1207.94,E2 -1207.94} C_VEL
LIN {X 0,Y 594.377,Z 244.068,A -85,B 0,C 180,E1 -1210.822,E2 -1210.822} C_VEL
LIN {X 0,Y 594.378,Z 244.068,A -85,B 0,C 180,E1 -1213.84,E2 -1213.84} C_VEL
LIN {X 0,Y 594.361,Z 244.072,A -85,B 0,C 180,E1 -1216.7,E2 -1216.7} C_VEL
LIN {X 0,Y 594.364,Z 244.067,A -85,B 0,C 180,E1 -1219.433,E2 -1219.433} C_VEL
LIN {X 0,Y 594.385,Z 244.071,A -85,B 0,C 180,E1 -1222.391,E2 -1222.391} C_VEL
LIN {X 0,Y 594.38,Z 244.065,A -85,B 0,C 180,E1 -1224.671,E2 -1224.671} C_VEL
LIN {X 0,Y 594.371,Z 244.065,A -85,B 0,C 180,E1 -1227.088,E2 -1227.088} C_VEL
LIN {X 0,Y 594.394,Z 244.068,A -85,B 0,C 180,E1 -1229.669,E2 -1229.669} C_VEL
LIN {X 0,Y 594.384,Z 244.067,A -85,B 0,C 180,E1 -1232.54,E2 -1232.54} C_VEL
LIN {X 0,Y 594.372,Z 244.067,A -85,B 0,C 180,E1 -1234.807,E2 -1234.807} C_VEL
LIN {X 0,Y 594.356,Z 244.069,A -85,B 0,C 180,E1 -1237.264,E2 -1237.264} C_VEL
LIN {X 0,Y 594.373,Z 244.076,A -85,B 0,C 180,E1 -1239.946,E2 -1239.946} C_VEL
LIN {X 0,Y 594.385,Z 244.064,A -85,B 0,C 180,E1 -1242.807,E2 -1242.807} C_VEL
LIN {X 0,Y 594.38,Z 244.075,A -85,B 0,C 180,E1 -1245.825,E2 -1245.825} C_VEL
LIN {X 0,Y 594.387,Z 244.065,A -85,B 0,C 180,E1 -1248.404,E2 -1248.404} C_VEL
LIN {X 0,Y 594.394,Z 244.066,A -85,B 0,C 180,E1 -1251.158,E2 -1251.158} C_VEL
LIN {X 0,Y 594.362,Z 244.073,A -85,B 0,C 180,E1 -1253.891,E2 -1253.891} C_VEL
LIN {X 0,Y 594.378,Z 244.065,A -85,B 0,C 180,E1 -1256.611,E2 -1256.611} C_VEL
LIN {X 0,Y 594.417,Z 244.068,A -85,B 0,C 180,E1 -1259.323,E2 -1259.323} C_VEL
LIN {X 0,Y 594.388,Z 244.065,A -85,B 0,C 180,E1 -1262.033,E2 -1262.033} C_VEL
LIN {X 0,Y 594.393,Z 244.065,A -85,B 0,C 180,E1 -1264.748,E2 -1264.748} C_VEL
LIN {X 0,Y 594.394,Z 244.072,A -85,B 0,C 180,E1 -1267.473,E2 -1267.473} C_VEL
LIN {X 0,Y 594.387,Z 244.064,A -85,B 0,C 180,E1 -1270.216,E2 -1270.216} C_VEL
LIN {X 0,Y 594.368,Z 244.072,A -85,B 0,C 180,E1 -1272.983,E2 -1272.983} C_VEL
LIN {X 0,Y 594.358,Z 244.072,A -85,B 0,C 180,E1 -1275.335,E2 -1275.335} C_VEL
LIN {X 0,Y 593.688,Z 244.154,A -85,B 0,C 180,E1 -1275.901,E2 -1275.901} C_VEL
LIN {X 0,Y 590.833,Z 244.511,A -85,B 0,C 180,E1 -1276.819,E2 -1276.819} C_VEL
LIN {X 0,Y 588.427,Z 244.812,A -85,B 0,C 180,E1 -1277.558,E2 -1277.558} C_VEL
LIN {X 0,Y 587.398,Z 244.936,A -85,B 0,C 180,E1 -1278.128,E2 -1278.128} C_VEL
LIN {X 0,Y 587.317,Z 244.946,A -85,B 0,C 180,E1 -1278.321,E2 -1278.321} C_VEL
LIN {X 0,Y 587.321,Z 244.953,A -85,B 0,C 180,E1 -1281.038,E2 -1281.038} C_VEL
LIN {X 0,Y 587.317,Z 244.953,A -85,B 0,C 180,E1 -1283.259,E2 -1283.259} C_VEL
LIN {X 0,Y 587.33,Z 244.946,A -85,B 0,C 180,E1 -1285.517,E2 -1285.517} C_VEL
LIN {X 0,Y 587.342,Z 244.943,A -85,B 0,C 180,E1 -1287.818,E2 -1287.818} C_VEL
LIN {X 0,Y 587.345,Z 244.945,A -85,B 0,C 180,E1 -1290.513,E2 -1290.513} C_VEL
LIN {X 0,Y 587.329,Z 244.943,A -85,B 0,C 180,E1 -1293.397,E2 -1293.397} C_VEL
LIN {X 0,Y 587.352,Z 244.94,A -85,B 0,C 180,E1 -1295.896,E2 -1295.896} C_VEL
LIN {X 0,Y 587.329,Z 244.949,A -85,B 0,C 180,E1 -1298.48,E2 -1298.48} C_VEL
LIN {X 0,Y 587.332,Z 244.945,A -85,B 0,C 180,E1 -1301.158,E2 -1301.158} C_VEL
LIN {X 0,Y 587.322,Z 244.946,A -85,B 0,C 180,E1 -1304.114,E2 -1304.114} C_VEL
LIN {X 0,Y 587.319,Z 244.948,A -85,B 0,C 180,E1 -1306.995,E2 -1306.995} C_VEL
LIN {X 0,Y 587.315,Z 244.946,A -85,B 0,C 180,E1 -1309.747,E2 -1309.747} C_VEL
LIN {X 0,Y 587.342,Z 244.949,A -85,B 0,C 180,E1 -1312.393,E2 -1312.393} C_VEL
LIN {X 0,Y 587.326,Z 244.947,A -85,B 0,C 180,E1 -1314.945,E2 -1314.945} C_VEL
LIN {X 0,Y 587.34,Z 244.943,A -85,B 0,C 180,E1 -1317.422,E2 -1317.422} C_VEL
LIN {X 0,Y 587.332,Z 244.946,A -85,B 0,C 180,E1 -1319.83,E2 -1319.83} C_VEL
LIN {X 0,Y 587.352,Z 244.948,A -85,B 0,C 180,E1 -1322.308,E2 -1322.308} C_VEL
LIN {X 0,Y 587.337,Z 244.949,A -85,B 0,C 180,E1 -1324.484,E2 -1324.484} C_VEL
LIN {X 0,Y 587.346,Z 244.949,A -85,B 0,C 180,E1 -1327.487,E2 -1327.487} C_VEL
LIN {X 0,Y 587.381,Z 245.224,A -85,B 0,C 180,E1 -1327.813,E2 -1327.813} C_VEL
LIN {X 0,Y 587.801,Z 249.25,A -85,B 0,C 180,E1 -1328.425,E2 -1328.425} C_VEL
LIN {X 0,Y 587.612,Z 268.36,A -85,B 0,C 180,E1 -1331.16,E2 -1331.16} C_VEL
LIN {X 0,Y 587.568,Z 286.334,A -85,B 0,C 180,E1 -1333.675,E2 -1333.675} C_VEL
LIN {X 0,Y 588.187,Z 290.4,A -85,B 0,C 180,E1 -1333.77,E2 -1333.77} C_VEL
LIN {X 0,Y 587.996,Z 423.858,A -85,B 0,C 180,E1 -1335.441,E2 -1335.441} C_VEL
LIN {X 0,Y 587.917,Z 438.136,A -85,B 0,C 180,E1 -1335.764,E2 -1335.764} C_VEL
LIN {X 0,Y 587.856,Z 451.691,A -85,B 0,C 180,E1 -1336.211,E2 -1336.211} C_VEL
LIN {X 0,Y 587.733,Z 464.75,A -85,B 0,C 180,E1 -1336.78,E2 -1336.78} C_VEL
LIN {X 0,Y 587.626,Z 477.379,A -85,B 0,C 180,E1 -1337.481,E2 -1337.481} C_VEL
LIN {X 0,Y 587.514,Z 488.882,A -85,B 0,C 180,E1 -1338.267,E2 -1338.267} C_VEL
LIN {X 0,Y 587.467,Z 499.436,A -85,B 0,C 180,E1 -1339.14,E2 -1339.14} C_VEL
LIN {X 0,Y 587.355,Z 509.915,A -85,B 0,C 180,E1 -1340.183,E2 -1340.183} C_VEL
LIN {X 0,Y 587.311,Z 518.563,A -85,B 0,C 180,E1 -1341.224,E2 -1341.224} C_VEL
LIN {X 0,Y 587.25,Z 526.85,A -85,B 0,C 180,E1 -1342.436,E2 -1342.436} C_VEL
LIN {X 0,Y 587.181,Z 533.471,A -85,B 0,C 180,E1 -1343.636,E2 -1343.636} C_VEL
LIN {X 0,Y 587.158,Z 538.794,A -85,B 0,C 180,E1 -1344.85,E2 -1344.85} C_VEL
LIN {X 0,Y 587.181,Z 542.305,A -85,B 0,C 180,E1 -1345.882,E2 -1345.882} C_VEL
LIN {X 0,Y 587.13,Z 545.739,A -85,B 0,C 180,E1 -1347.256,E2 -1347.256} C_VEL
LIN {X 0,Y 587.145,Z 547.781,A -85,B 0,C 180,E1 -1348.628,E2 -1348.628} C_VEL
LIN {X 0,Y 587.136,Z 548.496,A -85,B 0,C 180,E1 -1350,E2 -1350} C_VEL
LIN {X 0,Y 587.142,Z 547.881,A -85,B 0,C 180,E1 -1351.372,E2 -1351.372} C_VEL
LIN {X 0,Y 587.128,Z 545.926,A -85,B 0,C 180,E1 -1352.744,E2 -1352.744} C_VEL
LIN {X 0,Y 587.182,Z 542.581,A -85,B 0,C 180,E1 -1354.118,E2 -1354.118} C_VEL
LIN {X 0,Y 587.2,Z 537.755,A -85,B 0,C 180,E1 -1355.494,E2 -1355.494} C_VEL
LIN {X 0,Y 587.21,Z 531.29,A -85,B 0,C 180,E1 -1356.874,E2 -1356.874} C_VEL
LIN {X 0,Y 587.269,Z 524.092,A -85,B 0,C 180,E1 -1358.083,E2 -1358.083} C_VEL
LIN {X 0,Y 587.332,Z 516.554,A -85,B 0,C 180,E1 -1359.122,E2 -1359.122} C_VEL
LIN {X 0,Y 587.376,Z 507.503,A -85,B 0,C 180,E1 -1360.165,E2 -1360.165} C_VEL
LIN {X 0,Y 587.503,Z 496.548,A -85,B 0,C 180,E1 -1361.208,E2 -1361.208} C_VEL
LIN {X 0,Y 587.566,Z 485.369,A -85,B 0,C 180,E1 -1362.082,E2 -1362.082} C_VEL
LIN {X 0,Y 587.642,Z 473.023,A -85,B 0,C 180,E1 -1362.87,E2 -1362.87} C_VEL
LIN {X 0,Y 587.783,Z 461.148,A -85,B 0,C 180,E1 -1363.483,E2 -1363.483} C_VEL
LIN {X 0,Y 587.894,Z 447.805,A -85,B 0,C 180,E1 -1364.022,E2 -1364.022} C_VEL
LIN {X 0,Y 587.941,Z 433.913,A -85,B 0,C 180,E1 -1364.435,E2 -1364.435} C_VEL
LIN {X 0,Y 588.019,Z 419.704,A -85,B 0,C 180,E1 -1364.713,E2 -1364.713} C_VEL
LIN {X 0,Y 588.111,Z 289.675,A -85,B 0,C 180,E1 -1366.332,E2 -1366.332} C_VEL
LIN {X 0,Y 587.556,Z 286.34,A -85,B 0,C 180,E1 -1366.414,E2 -1366.414} C_VEL
LIN {X 0,Y 587.673,Z 266.925,A -85,B 0,C 180,E1 -1369.132,E2 -1369.132} C_VEL
LIN {X 0,Y 587.834,Z 248.628,A -85,B 0,C 180,E1 -1371.754,E2 -1371.754} C_VEL
LIN {X 0,Y 587.371,Z 245.064,A -85,B 0,C 180,E1 -1372.327,E2 -1372.327} C_VEL
LIN {X 0,Y 587.351,Z 244.941,A -85,B 0,C 180,E1 -1374.758,E2 -1374.758} C_VEL
LIN {X 0,Y 587.327,Z 244.946,A -85,B 0,C 180,E1 -1377.046,E2 -1377.046} C_VEL
LIN {X 0,Y 587.347,Z 244.946,A -85,B 0,C 180,E1 -1379.379,E2 -1379.379} C_VEL
LIN {X 0,Y 587.345,Z 244.949,A -85,B 0,C 180,E1 -1381.835,E2 -1381.835} C_VEL
LIN {X 0,Y 587.346,Z 244.942,A -85,B 0,C 180,E1 -1384.347,E2 -1384.347} C_VEL
LIN {X 0,Y 587.35,Z 244.942,A -85,B 0,C 180,E1 -1386.746,E2 -1386.746} C_VEL
LIN {X 0,Y 587.339,Z 244.95,A -85,B 0,C 180,E1 -1389.359,E2 -1389.359} C_VEL
LIN {X 0,Y 587.331,Z 244.943,A -85,B 0,C 180,E1 -1392.107,E2 -1392.107} C_VEL
LIN {X 0,Y 587.312,Z 244.951,A -85,B 0,C 180,E1 -1395.088,E2 -1395.088} C_VEL
LIN {X 0,Y 587.348,Z 244.941,A -85,B 0,C 180,E1 -1397.927,E2 -1397.927} C_VEL
LIN {X 0,Y 587.329,Z 244.95,A -85,B 0,C 180,E1 -1401.057,E2 -1401.057} C_VEL
LIN {X 0,Y 587.348,Z 244.951,A -85,B 0,C 180,E1 -1403.291,E2 -1403.291} C_VEL
LIN {X 0,Y 587.364,Z 244.938,A -85,B 0,C 180,E1 -1405.78,E2 -1405.78} C_VEL
LIN {X 0,Y 587.345,Z 244.94,A -85,B 0,C 180,E1 -1408.231,E2 -1408.231} C_VEL
LIN {X 0,Y 587.344,Z 244.948,A -85,B 0,C 180,E1 -1410.865,E2 -1410.865} C_VEL
LIN {X 0,Y 587.351,Z 244.941,A -85,B 0,C 180,E1 -1413.818,E2 -1413.818} C_VEL
LIN {X 0,Y 587.333,Z 244.944,A -85,B 0,C 180,E1 -1415.993,E2 -1415.993} C_VEL
LIN {X 0,Y 587.316,Z 244.946,A -85,B 0,C 180,E1 -1418.225,E2 -1418.225} C_VEL
LIN {X 0,Y 587.343,Z 244.948,A -85,B 0,C 180,E1 -1421.151,E2 -1421.151} C_VEL
LIN {X 0,Y 587.346,Z 244.944,A -85,B 0,C 180,E1 -1423.311,E2 -1423.311} C_VEL
LIN {X 0,Y 587.354,Z 244.941,A -85,B 0,C 180,E1 -1426.154,E2 -1426.154} C_VEL
LIN {X 0,Y 587.337,Z 244.949,A -85,B 0,C 180,E1 -1428.962,E2 -1428.962} C_VEL
LIN {X 0,Y 587.362,Z 244.939,A -85,B 0,C 180,E1 -1431.745,E2 -1431.745} C_VEL
LIN {X 0,Y 587.356,Z 244.949,A -85,B 0,C 180,E1 -1434.507,E2 -1434.507} C_VEL
LIN {X 0,Y 587.373,Z 244.938,A -85,B 0,C 180,E1 -1437.257,E2 -1437.257} C_VEL
LIN {X 0,Y 587.373,Z 244.941,A -85,B 0,C 180,E1 -1440,E2 -1440} C_VEL
LIN {X 0,Y 587.373,Z 244.943,A -85,B 0,C 180,E1 -1442.743,E2 -1442.743} C_VEL
LIN {X 0,Y 587.354,Z 244.94,A -85,B 0,C 180,E1 -1445.493,E2 -1445.493} C_VEL
LIN {X 0,Y 587.363,Z 244.948,A -85,B 0,C 180,E1 -1448.255,E2 -1448.255} C_VEL
LIN {X 0,Y 587.337,Z 244.943,A -85,B 0,C 180,E1 -1451.134,E2 -1451.134} C_VEL
LIN {X 0,Y 587.354,Z 244.944,A -85,B 0,C 180,E1 -1453.846,E2 -1453.846} C_VEL
LIN {X 0,Y 587.354,Z 244.942,A -85,B 0,C 180,E1 -1456.82,E2 -1456.82} C_VEL
LIN {X 0,Y 587.338,Z 244.945,A -85,B 0,C 180,E1 -1459.575,E2 -1459.575} C_VEL
LIN {X 0,Y 587.332,Z 244.947,A -85,B 0,C 180,E1 -1462.514,E2 -1462.514} C_VEL
LIN {X 0,Y 587.344,Z 244.943,A -85,B 0,C 180,E1 -1464.759,E2 -1464.759} C_VEL
LIN {X 0,Y 587.332,Z 244.943,A -85,B 0,C 180,E1 -1467.046,E2 -1467.046} C_VEL
LIN {X 0,Y 587.344,Z 244.944,A -85,B 0,C 180,E1 -1469.38,E2 -1469.38} C_VEL
LIN {X 0,Y 587.347,Z 244.95,A -85,B 0,C 180,E1 -1471.838,E2 -1471.838} C_VEL
LIN {X 0,Y 587.35,Z 244.941,A -85,B 0,C 180,E1 -1474.35,E2 -1474.35} C_VEL
LIN {X 0,Y 587.347,Z 244.941,A -85,B 0,C 180,E1 -1476.747,E2 -1476.747} C_VEL
LIN {X 0,Y 587.342,Z 244.946,A -85,B 0,C 180,E1 -1479.36,E2 -1479.36} C_VEL
LIN {X 0,Y 587.329,Z 244.948,A -85,B 0,C 180,E1 -1482.108,E2 -1482.108} C_VEL
LIN {X 0,Y 587.311,Z 244.948,A -85,B 0,C 180,E1 -1485.089,E2 -1485.089} C_VEL
LIN {X 0,Y 587.348,Z 244.945,A -85,B 0,C 180,E1 -1487.928,E2 -1487.928} C_VEL
LIN {X 0,Y 587.329,Z 244.947,A -85,B 0,C 180,E1 -1491.059,E2 -1491.059} C_VEL
LIN {X 0,Y 587.344,Z 244.947,A -85,B 0,C 180,E1 -1493.293,E2 -1493.293} C_VEL
LIN {X 0,Y 587.363,Z 244.944,A -85,B 0,C 180,E1 -1495.781,E2 -1495.781} C_VEL
LIN {X 0,Y 587.351,Z 244.942,A -85,B 0,C 180,E1 -1498.233,E2 -1498.233} C_VEL
LIN {X 0,Y 587.349,Z 244.941,A -85,B 0,C 180,E1 -1500.867,E2 -1500.867} C_VEL
LIN {X 0,Y 587.359,Z 244.943,A -85,B 0,C 180,E1 -1503.819,E2 -1503.819} C_VEL
LIN {X 0,Y 587.357,Z 245.076,A -85,B 0,C 180,E1 -1506.697,E2 -1506.697} C_VEL
LIN {X 0,Y 587.926,Z 249.215,A -85,B 0,C 180,E1 -1507.333,E2 -1507.333} C_VEL
LIN {X 0,Y 587.719,Z 271.987,A -85,B 0,C 180,E1 -1510.439,E2 -1510.439} C_VEL
LIN {X 0,Y 587.56,Z 293.471,A -85,B 0,C 180,E1 -1513.318,E2 -1513.318} C_VEL
LIN {X 0,Y 587.584,Z 296.198,A -85,B 0,C 180,E1 -1513.642,E2 -1513.642} C_VEL
LIN {X 0,Y 588.193,Z 299.646,A -85,B 0,C 180,E1 -1513.715,E2 -1513.715} C_VEL
LIN {X 0,Y 587.988,Z 433.904,A -85,B 0,C 180,E1 -1515.397,E2 -1515.397} C_VEL
LIN {X 0,Y 587.947,Z 448.255,A -85,B 0,C 180,E1 -1515.723,E2 -1515.723} C_VEL
LIN {X 0,Y 587.817,Z 461.721,A -85,B 0,C 180,E1 -1516.166,E2 -1516.166} C_VEL
LIN {X 0,Y 587.731,Z 475.646,A -85,B 0,C 180,E1 -1516.78,E2 -1516.78} C_VEL
LIN {X 0,Y 587.605,Z 488.103,A -85,B 0,C 180,E1 -1517.48,E2 -1517.48} C_VEL
LIN {X 0,Y 587.513,Z 500.643,A -85,B 0,C 180,E1 -1518.354,E2 -1518.354} C_VEL
LIN {X 0,Y 587.444,Z 511.838,A -85,B 0,C 180,E1 -1519.314,E2 -1519.314} C_VEL
LIN {X 0,Y 587.319,Z 521.853,A -85,B 0,C 180,E1 -1520.356,E2 -1520.356} C_VEL
LIN {X 0,Y 587.277,Z 530.173,A -85,B 0,C 180,E1 -1521.397,E2 -1521.397} C_VEL
LIN {X 0,Y 587.244,Z 538.127,A -85,B 0,C 180,E1 -1522.608,E2 -1522.608} C_VEL
LIN {X 0,Y 587.204,Z 544.528,A -85,B 0,C 180,E1 -1523.816,E2 -1523.816} C_VEL
LIN {X 0,Y 587.16,Z 548.962,A -85,B 0,C 180,E1 -1524.85,E2 -1524.85} C_VEL
LIN {X 0,Y 587.179,Z 552.443,A -85,B 0,C 180,E1 -1525.882,E2 -1525.882} C_VEL
LIN {X 0,Y 587.13,Z 555.832,A -85,B 0,C 180,E1 -1527.256,E2 -1527.256} C_VEL
LIN {X 0,Y 587.142,Z 557.832,A -85,B 0,C 180,E1 -1528.628,E2 -1528.628} C_VEL
LIN {X 0,Y 587.135,Z 558.5,A -85,B 0,C 180,E1 -1530,E2 -1530} C_VEL
LIN {X 0,Y 587.142,Z 557.832,A -85,B 0,C 180,E1 -1531.372,E2 -1531.372} C_VEL
LIN {X 0,Y 587.13,Z 555.833,A -85,B 0,C 180,E1 -1532.744,E2 -1532.744} C_VEL
LIN {X 0,Y 587.179,Z 552.444,A -85,B 0,C 180,E1 -1534.118,E2 -1534.118} C_VEL
LIN {X 0,Y 587.2,Z 547.568,A -85,B 0,C 180,E1 -1535.494,E2 -1535.494} C_VEL
LIN {X 0,Y 587.209,Z 541.053,A -85,B 0,C 180,E1 -1536.874,E2 -1536.874} C_VEL
LIN {X 0,Y 587.268,Z 533.8,A -85,B 0,C 180,E1 -1538.083,E2 -1538.083} C_VEL
LIN {X 0,Y 587.321,Z 524.824,A -85,B 0,C 180,E1 -1539.296,E2 -1539.296} C_VEL
LIN {X 0,Y 587.372,Z 515.393,A -85,B 0,C 180,E1 -1540.339,E2 -1540.339} C_VEL
LIN {X 0,Y 587.475,Z 505.029,A -85,B 0,C 180,E1 -1541.29,E2 -1541.29} C_VEL
LIN {X 0,Y 587.577,Z 493.434,A -85,B 0,C 180,E1 -1542.17,E2 -1542.17} C_VEL
LIN {X 0,Y 587.67,Z 480.652,A -85,B 0,C 180,E1 -1542.958,E2 -1542.958} C_VEL
LIN {X 0,Y 587.799,Z 468.164,A -85,B 0,C 180,E1 -1543.57,E2 -1543.57} C_VEL
LIN {X 0,Y 587.916,Z 454.613,A -85,B 0,C 180,E1 -1544.085,E2 -1544.085} C_VEL
LIN {X 0,Y 587.986,Z 440.73,A -85,B 0,C 180,E1 -1544.466,E2 -1544.466} C_VEL
LIN {X 0,Y 588.019,Z 426.622,A -85,B 0,C 180,E1 -1544.713,E2 -1544.713} C_VEL
LIN {X 0,Y 588.107,Z 299.193,A -85,B 0,C 180,E1 -1546.293,E2 -1546.293} C_VEL
LIN {X 0,Y 587.586,Z 296.007,A -85,B 0,C 180,E1 -1546.369,E2 -1546.369} C_VEL
LIN {X 0,Y 587.61,Z 276.17,A -85,B 0,C 180,E1 -1549,E2 -1549} C_VEL
LIN {X 0,Y 587.769,Z 260.315,A -85,B 0,C 180,E1 -1551.148,E2 -1551.148} C_VEL
LIN {X 0,Y 587.942,Z 248.787,A -85,B 0,C 180,E1 -1552.726,E2 -1552.726} C_VEL
LIN {X 0,Y 587.357,Z 245.075,A -85,B 0,C 180,E1 -1553.303,E2 -1553.303} C_VEL
LIN {X 0,Y 587.359,Z 244.943,A -85,B 0,C 180,E1 -1556.181,E2 -1556.181} C_VEL
LIN {X 0,Y 587.349,Z 244.941,A -85,B 0,C 180,E1 -1559.133,E2 -1559.133} C_VEL
LIN {X 0,Y 587.347,Z 244.943,A -85,B 0,C 180,E1 -1561.836,E2 -1561.836} C_VEL
LIN {X 0,Y 587.347,Z 244.948,A -85,B 0,C 180,E1 -1564.347,E2 -1564.347} C_VEL
LIN {X 0,Y 587.341,Z 244.942,A -85,B 0,C 180,E1 -1567.607,E2 -1567.607} C_VEL
LIN {X 0,Y 587.31,Z 244.954,A -85,B 0,C 180,E1 -1570.254,E2 -1570.254} C_VEL
LIN {X 0,Y 587.32,Z 244.946,A -85,B 0,C 180,E1 -1573.005,E2 -1573.005} C_VEL
LIN {X 0,Y 587.321,Z 244.948,A -85,B 0,C 180,E1 -1575.886,E2 -1575.886} C_VEL
LIN {X 0,Y 587.332,Z 244.944,A -85,B 0,C 180,E1 -1578.924,E2 -1578.924} C_VEL
LIN {X 0,Y 587.329,Z 244.945,A -85,B 0,C 180,E1 -1581.521,E2 -1581.521} C_VEL
LIN {X 0,Y 587.347,Z 244.943,A -85,B 0,C 180,E1 -1584.454,E2 -1584.454} C_VEL
LIN {X 0,Y 587.332,Z 244.942,A -85,B 0,C 180,E1 -1586.888,E2 -1586.888} C_VEL
LIN {X 0,Y 587.344,Z 244.944,A -85,B 0,C 180,E1 -1589.487,E2 -1589.487} C_VEL
LIN {X 0,Y 587.344,Z 244.947,A -85,B 0,C 180,E1 -1592.306,E2 -1592.306} C_VEL
LIN {X 0,Y 587.33,Z 244.946,A -85,B 0,C 180,E1 -1594.483,E2 -1594.483} C_VEL
LIN {X 0,Y 587.311,Z 244.946,A -85,B 0,C 180,E1 -1597.131,E2 -1597.131} C_VEL
LIN {X 0,Y 587.325,Z 244.951,A -85,B 0,C 180,E1 -1599.695,E2 -1599.695} C_VEL
LIN {X 0,Y 587.352,Z 244.941,A -85,B 0,C 180,E1 -1602.594,E2 -1602.594} C_VEL
LIN {X 0,Y 587.356,Z 244.95,A -85,B 0,C 180,E1 -1605.739,E2 -1605.739} C_VEL
LIN {X 0,Y 587.335,Z 244.945,A -85,B 0,C 180,E1 -1608.263,E2 -1608.263} C_VEL
LIN {X 0,Y 587.339,Z 244.943,A -85,B 0,C 180,E1 -1611.051,E2 -1611.051} C_VEL
LIN {X 0,Y 587.366,Z 244.944,A -85,B 0,C 180,E1 -1613.264,E2 -1613.264} C_VEL
LIN {X 0,Y 587.31,Z 244.95,A -85,B 0,C 180,E1 -1615.883,E2 -1615.883} C_VEL
LIN {X 0,Y 587.359,Z 244.944,A -85,B 0,C 180,E1 -1617.943,E2 -1617.943} C_VEL
LIN {X 0,Y 587.387,Z 244.937,A -85,B 0,C 180,E1 -1620.686,E2 -1620.686} C_VEL
LIN {X 0,Y 587.33,Z 244.952,A -85,B 0,C 180,E1 -1623.43,E2 -1623.43} C_VEL
LIN {X 0,Y 587.354,Z 244.95,A -85,B 0,C 180,E1 -1625.493,E2 -1625.493} C_VEL
LIN {X 0,Y 587.363,Z 244.939,A -85,B 0,C 180,E1 -1628.255,E2 -1628.255} C_VEL
LIN {X 0,Y 587.338,Z 244.95,A -85,B 0,C 180,E1 -1631.134,E2 -1631.134} C_VEL
LIN {X 0,Y 587.354,Z 244.942,A -85,B 0,C 180,E1 -1633.846,E2 -1633.846} C_VEL
LIN {X 0,Y 587.355,Z 244.944,A -85,B 0,C 180,E1 -1636.82,E2 -1636.82} C_VEL
LIN {X 0,Y 587.317,Z 244.946,A -85,B 0,C 180,E1 -1638.321,E2 -1638.321} C_VEL
LIN {X 0,Y 586.663,Z 245.034,A -85,B 0,C 180,E1 -1638.893,E2 -1638.893} C_VEL
LIN {X 0,Y 583.83,Z 245.391,A -85,B 0,C 180,E1 -1639.821,E2 -1639.821} C_VEL
LIN {X 0,Y 581.419,Z 245.693,A -85,B 0,C 180,E1 -1640.568,E2 -1640.568} C_VEL
LIN {X 0,Y 580.368,Z 245.82,A -85,B 0,C 180,E1 -1641.144,E2 -1641.144} C_VEL
LIN {X 0,Y 580.274,Z 245.829,A -85,B 0,C 180,E1 -1641.34,E2 -1641.34} C_VEL
LIN {X 0,Y 580.295,Z 245.821,A -85,B 0,C 180,E1 -1644.317,E2 -1644.317} C_VEL
LIN {X 0,Y 580.275,Z 245.825,A -85,B 0,C 180,E1 -1646.624,E2 -1646.624} C_VEL
LIN {X 0,Y 580.299,Z 245.824,A -85,B 0,C 180,E1 -1649.311,E2 -1649.311} C_VEL
LIN {X 0,Y 580.296,Z 245.818,A -85,B 0,C 180,E1 -1652.201,E2 -1652.201} C_VEL
LIN {X 0,Y 580.297,Z 245.823,A -85,B 0,C 180,E1 -1654.696,E2 -1654.696} C_VEL
LIN {X 0,Y 580.295,Z 245.824,A -85,B 0,C 180,E1 -1657.269,E2 -1657.269} C_VEL
LIN {X 0,Y 580.294,Z 245.822,A -85,B 0,C 180,E1 -1660.272,E2 -1660.272} C_VEL
LIN {X 0,Y 580.273,Z 245.829,A -85,B 0,C 180,E1 -1662.707,E2 -1662.707} C_VEL
LIN {X 0,Y 580.271,Z 245.823,A -85,B 0,C 180,E1 -1665.609,E2 -1665.609} C_VEL
LIN {X 0,Y 580.311,Z 245.819,A -85,B 0,C 180,E1 -1668.235,E2 -1668.235} C_VEL
LIN {X 0,Y 580.28,Z 245.826,A -85,B 0,C 180,E1 -1670.966,E2 -1670.966} C_VEL
LIN {X 0,Y 580.28,Z 245.822,A -85,B 0,C 180,E1 -1673.598,E2 -1673.598} C_VEL
LIN {X 0,Y 580.316,Z 245.822,A -85,B 0,C 180,E1 -1676.146,E2 -1676.146} C_VEL
LIN {X 0,Y 580.277,Z 245.83,A -85,B 0,C 180,E1 -1678.615,E2 -1678.615} C_VEL
LIN {X 0,Y 580.293,Z 245.821,A -85,B 0,C 180,E1 -1681.025,E2 -1681.025} C_VEL
LIN {X 0,Y 580.293,Z 245.823,A -85,B 0,C 180,E1 -1683.666,E2 -1683.666} C_VEL
LIN {X 0,Y 580.301,Z 245.821,A -85,B 0,C 180,E1 -1685.684,E2 -1685.684} C_VEL
LIN {X 0,Y 580.342,Z 246.058,A -85,B 0,C 180,E1 -1687.646,E2 -1687.646} C_VEL
LIN {X 0,Y 580.875,Z 250.557,A -85,B 0,C 180,E1 -1688.346,E2 -1688.346} C_VEL
LIN {X 0,Y 580.662,Z 269.636,A -85,B 0,C 180,E1 -1691.11,E2 -1691.11} C_VEL
LIN {X 0,Y 580.562,Z 286.353,A -85,B 0,C 180,E1 -1693.473,E2 -1693.473} C_VEL
LIN {X 0,Y 581.388,Z 291.44,A -85,B 0,C 180,E1 -1693.587,E2 -1693.587} C_VEL
LIN {X 0,Y 581.141,Z 423.887,A -85,B 0,C 180,E1 -1695.266,E2 -1695.266} C_VEL
LIN {X 0,Y 581.05,Z 438.132,A -85,B 0,C 180,E1 -1695.592,E2 -1695.592} C_VEL
LIN {X 0,Y 580.938,Z 451.703,A -85,B 0,C 180,E1 -1696.043,E2 -1696.043} C_VEL
LIN {X 0,Y 580.804,Z 464.759,A -85,B 0,C 180,E1 -1696.619,E2 -1696.619} C_VEL
LIN {X 0,Y 580.66,Z 477.39,A -85,B 0,C 180,E1 -1697.328,E2 -1697.328} C_VEL
LIN {X 0,Y 580.542,Z 488.892,A -85,B 0,C 180,E1 -1698.124,E2 -1698.124} C_VEL
LIN {X 0,Y 580.462,Z 499.455,A -85,B 0,C 180,E1 -1699.008,E2 -1699.008} C_VEL
LIN {X 0,Y 580.318,Z 509.92,A -85,B 0,C 180,E1 -1700.063,E2 -1700.063} C_VEL
LIN {X 0,Y 580.254,Z 518.567,A -85,B 0,C 180,E1 -1701.117,E2 -1701.117} C_VEL
LIN {X 0,Y 580.176,Z 526.854,A -85,B 0,C 180,E1 -1702.343,E2 -1702.343} C_VEL
LIN {X 0,Y 580.124,Z 532.757,A -85,B 0,C 180,E1 -1703.416,E2 -1703.416} C_VEL
LIN {X 0,Y 580.129,Z 537.385,A -85,B 0,C 180,E1 -1704.438,E2 -1704.438} C_VEL
LIN {X 0,Y 580.103,Z 542.307,A -85,B 0,C 180,E1 -1705.832,E2 -1705.832} C_VEL
LIN {X 0,Y 580.041,Z 545.74,A -85,B 0,C 180,E1 -1707.222,E2 -1707.222} C_VEL
LIN {X 0,Y 580.045,Z 547.782,A -85,B 0,C 180,E1 -1708.611,E2 -1708.611} C_VEL
LIN {X 0,Y 580.037,Z 548.496,A -85,B 0,C 180,E1 -1710,E2 -1710} C_VEL
LIN {X 0,Y 580.042,Z 547.881,A -85,B 0,C 180,E1 -1711.388,E2 -1711.388} C_VEL
LIN {X 0,Y 580.039,Z 545.925,A -85,B 0,C 180,E1 -1712.778,E2 -1712.778} C_VEL
LIN {X 0,Y 580.104,Z 542.58,A -85,B 0,C 180,E1 -1714.168,E2 -1714.168} C_VEL
LIN {X 0,Y 580.129,Z 537.753,A -85,B 0,C 180,E1 -1715.561,E2 -1715.561} C_VEL
LIN {X 0,Y 580.142,Z 531.287,A -85,B 0,C 180,E1 -1716.958,E2 -1716.958} C_VEL
LIN {X 0,Y 580.192,Z 524.089,A -85,B 0,C 180,E1 -1718.182,E2 -1718.182} C_VEL
LIN {X 0,Y 580.284,Z 516.551,A -85,B 0,C 180,E1 -1719.234,E2 -1719.234} C_VEL
LIN {X 0,Y 580.347,Z 507.498,A -85,B 0,C 180,E1 -1720.289,E2 -1720.289} C_VEL
LIN {X 0,Y 580.494,Z 496.541,A -85,B 0,C 180,E1 -1721.346,E2 -1721.346} C_VEL
LIN {X 0,Y 580.575,Z 485.363,A -85,B 0,C 180,E1 -1722.23,E2 -1722.23} C_VEL
LIN {X 0,Y 580.706,Z 473.015,A -85,B 0,C 180,E1 -1723.027,E2 -1723.027} C_VEL
LIN {X 0,Y 580.873,Z 461.138,A -85,B 0,C 180,E1 -1723.646,E2 -1723.646} C_VEL
LIN {X 0,Y 581.002,Z 448.158,A -85,B 0,C 180,E1 -1724.179,E2 -1724.179} C_VEL
LIN {X 0,Y 581.07,Z 433.966,A -85,B 0,C 180,E1 -1724.608,E2 -1724.608} C_VEL
LIN {X 0,Y 581.161,Z 419.665,A -85,B 0,C 180,E1 -1724.89,E2 -1724.89} C_VEL
LIN {X 0,Y 581.316,Z 290.621,A -85,B 0,C 180,E1 -1726.515,E2 -1726.515} C_VEL
LIN {X 0,Y 580.579,Z 286.34,A -85,B 0,C 180,E1 -1726.617,E2 -1726.617} C_VEL
LIN {X 0,Y 580.7,Z 267.659,A -85,B 0,C 180,E1 -1729.264,E2 -1729.264} C_VEL
LIN {X 0,Y 580.901,Z 250.024,A -85,B 0,C 180,E1 -1731.821,E2 -1731.821} C_VEL
LIN {X 0,Y 580.329,Z 245.967,A -85,B 0,C 180,E1 -1732.472,E2 -1732.472} C_VEL
LIN {X 0,Y 580.307,Z 245.82,A -85,B 0,C 180,E1 -1735.079,E2 -1735.079} C_VEL
LIN {X 0,Y 580.301,Z 245.821,A -85,B 0,C 180,E1 -1738.185,E2 -1738.185} C_VEL
LIN {X 0,Y 580.282,Z 245.823,A -85,B 0,C 180,E1 -1740.694,E2 -1740.694} C_VEL
LIN {X 0,Y 580.303,Z 245.825,A -85,B 0,C 180,E1 -1743.316,E2 -1743.316} C_VEL
LIN {X 0,Y 580.274,Z 245.83,A -85,B 0,C 180,E1 -1745.76,E2 -1745.76} C_VEL
LIN {X 0,Y 580.285,Z 245.822,A -85,B 0,C 180,E1 -1748.146,E2 -1748.146} C_VEL
LIN {X 0,Y 580.296,Z 245.822,A -85,B 0,C 180,E1 -1750.842,E2 -1750.842} C_VEL
LIN {X 0,Y 580.284,Z 245.828,A -85,B 0,C 180,E1 -1753.656,E2 -1753.656} C_VEL
LIN {X 0,Y 580.272,Z 245.824,A -85,B 0,C 180,E1 -1756.609,E2 -1756.609} C_VEL
LIN {X 0,Y 580.294,Z 245.824,A -85,B 0,C 180,E1 -1759.156,E2 -1759.156} C_VEL
LIN {X 0,Y 580.285,Z 245.823,A -85,B 0,C 180,E1 -1761.926,E2 -1761.926} C_VEL
LIN {X 0,Y 580.302,Z 245.819,A -85,B 0,C 180,E1 -1764.456,E2 -1764.456} C_VEL
LIN {X 0,Y 580.284,Z 245.825,A -85,B 0,C 180,E1 -1766.975,E2 -1766.975} C_VEL
LIN {X 0,Y 580.304,Z 245.824,A -85,B 0,C 180,E1 -1769.425,E2 -1769.425} C_VEL
LIN {X 0,Y 580.312,Z 245.818,A -85,B 0,C 180,E1 -1772.136,E2 -1772.136} C_VEL
LIN {X 0,Y 580.314,Z 245.824,A -85,B 0,C 180,E1 -1775.269,E2 -1775.269} C_VEL
LIN {X 0,Y 580.266,Z 245.823,A -85,B 0,C 180,E1 -1777.947,E2 -1777.947} C_VEL
LIN {X 0,Y 580.309,Z 245.828,A -85,B 0,C 180,E1 -1780.914,E2 -1780.914} C_VEL
LIN {X 0,Y 580.276,Z 245.822,A -85,B 0,C 180,E1 -1783.825,E2 -1783.825} C_VEL
LIN {X 0,Y 580.275,Z 245.83,A -85,B 0,C 180,E1 -1786.696,E2 -1786.696} C_VEL
LIN {X 0,Y 580.295,Z 245.82,A -85,B 0,C 180,E1 -1789.533,E2 -1789.533} C_VEL
LIN {X 0,Y 580.324,Z 245.82,A -85,B 0,C 180,E1 -1792.345,E2 -1792.345} C_VEL
LIN {X 0,Y 580.333,Z 245.818,A -85,B 0,C 180,E1 -1795.137,E2 -1795.137} C_VEL
LIN {X 0,Y 580.328,Z 245.815,A -85,B 0,C 180,E1 -1797.918,E2 -1797.918} C_VEL
LIN {X 0,Y 580.359,Z 245.819,A -85,B 0,C 180,E1 -1800.694,E2 -1800.694} C_VEL
LIN {X 0,Y 580.281,Z 245.82,A -85,B 0,C 180,E1 -1803.472,E2 -1803.472} C_VEL
LIN {X 0,Y 580.319,Z 245.817,A -85,B 0,C 180,E1 -1805.56,E2 -1805.56} C_VEL
LIN {X 0,Y 580.327,Z 245.826,A -85,B 0,C 180,E1 -1808.356,E2 -1808.356} C_VEL
LIN {X 0,Y 580.289,Z 245.82,A -85,B 0,C 180,E1 -1811.191,E2 -1811.191} C_VEL
LIN {X 0,Y 580.318,Z 245.823,A -85,B 0,C 180,E1 -1814.017,E2 -1814.017} C_VEL
LIN {X 0,Y 580.305,Z 245.819,A -85,B 0,C 180,E1 -1816.915,E2 -1816.915} C_VEL
LIN {X 0,Y 580.3,Z 245.824,A -85,B 0,C 180,E1 -1819.822,E2 -1819.822} C_VEL
LIN {X 0,Y 580.287,Z 245.821,A -85,B 0,C 180,E1 -1822.803,E2 -1822.803} C_VEL
LIN {X 0,Y 580.299,Z 245.82,A -85,B 0,C 180,E1 -1825.08,E2 -1825.08} C_VEL
LIN {X 0,Y 580.294,Z 245.827,A -85,B 0,C 180,E1 -1828.186,E2 -1828.186} C_VEL
LIN {X 0,Y 580.292,Z 245.821,A -85,B 0,C 180,E1 -1830.698,E2 -1830.698} C_VEL
LIN {X 0,Y 580.297,Z 245.819,A -85,B 0,C 180,E1 -1833.317,E2 -1833.317} C_VEL
LIN {X 0,Y 580.32,Z 245.822,A -85,B 0,C 180,E1 -1835.768,E2 -1835.768} C_VEL
LIN {X 0,Y 580.283,Z 245.827,A -85,B 0,C 180,E1 -1838.147,E2 -1838.147} C_VEL
LIN {X 0,Y 580.295,Z 245.82,A -85,B 0,C 180,E1 -1840.844,E2 -1840.844} C_VEL
LIN {X 0,Y 580.273,Z 245.833,A -85,B 0,C 180,E1 -1843.658,E2 -1843.658} C_VEL
LIN {X 0,Y 580.288,Z 245.821,A -85,B 0,C 180,E1 -1846.608,E2 -1846.608} C_VEL
LIN {X 0,Y 580.297,Z 245.821,A -85,B 0,C 180,E1 -1849.158,E2 -1849.158} C_VEL
LIN {X 0,Y 580.286,Z 245.824,A -85,B 0,C 180,E1 -1851.928,E2 -1851.928} C_VEL
LIN {X 0,Y 580.253,Z 245.826,A -85,B 0,C 180,E1 -1854.454,E2 -1854.454} C_VEL
LIN {X 0,Y 580.29,Z 245.823,A -85,B 0,C 180,E1 -1856.976,E2 -1856.976} C_VEL
LIN {X 0,Y 580.299,Z 245.825,A -85,B 0,C 180,E1 -1859.426,E2 -1859.426} C_VEL
LIN {X 0,Y 580.296,Z 245.822,A -85,B 0,C 180,E1 -1862.142,E2 -1862.142} C_VEL
LIN {X 0,Y 580.321,Z 245.827,A -85,B 0,C 180,E1 -1865.27,E2 -1865.27} C_VEL
LIN {X 0,Y 580.358,Z 246.026,A -85,B 0,C 180,E1 -1866.548,E2 -1866.548} C_VEL
LIN {X 0,Y 581.022,Z 250.503,A -85,B 0,C 180,E1 -1867.228,E2 -1867.228} C_VEL
LIN {X 0,Y 580.782,Z 273.21,A -85,B 0,C 180,E1 -1870.363,E2 -1870.363} C_VEL
LIN {X 0,Y 580.569,Z 294.814,A -85,B 0,C 180,E1 -1873.292,E2 -1873.292} C_VEL
LIN {X 0,Y 580.648,Z 296.49,A -85,B 0,C 180,E1 -1873.453,E2 -1873.453} C_VEL
LIN {X 0,Y 581.394,Z 301.436,A -85,B 0,C 180,E1 -1873.542,E2 -1873.542} C_VEL
LIN {X 0,Y 581.138,Z 433.904,A -85,B 0,C 180,E1 -1875.221,E2 -1875.221} C_VEL
LIN {X 0,Y 581.075,Z 448.013,A -85,B 0,C 180,E1 -1875.544,E2 -1875.544} C_VEL
LIN {X 0,Y 580.914,Z 461.72,A -85,B 0,C 180,E1 -1875.998,E2 -1875.998} C_VEL
LIN {X 0,Y 580.791,Z 475.649,A -85,B 0,C 180,E1 -1876.619,E2 -1876.619} C_VEL
LIN {X 0,Y 580.656,Z 488.105,A -85,B 0,C 180,E1 -1877.328,E2 -1877.328} C_VEL
LIN {X 0,Y 580.524,Z 500.645,A -85,B 0,C 180,E1 -1878.212,E2 -1878.212} C_VEL
LIN {X 0,Y 580.441,Z 511.894,A -85,B 0,C 180,E1 -1879.189,E2 -1879.189} C_VEL
LIN {X 0,Y 580.276,Z 521.853,A -85,B 0,C 180,E1 -1880.238,E2 -1880.238} C_VEL
LIN {X 0,Y 580.241,Z 530.173,A -85,B 0,C 180,E1 -1881.292,E2 -1881.292} C_VEL
LIN {X 0,Y 580.165,Z 538.128,A -85,B 0,C 180,E1 -1882.518,E2 -1882.518} C_VEL
LIN {X 0,Y 580.103,Z 544.528,A -85,B 0,C 180,E1 -1883.74,E2 -1883.74} C_VEL
LIN {X 0,Y 580.078,Z 548.962,A -85,B 0,C 180,E1 -1884.787,E2 -1884.787} C_VEL
LIN {X 0,Y 580.102,Z 552.443,A -85,B 0,C 180,E1 -1885.832,E2 -1885.832} C_VEL
LIN {X 0,Y 580.041,Z 555.832,A -85,B 0,C 180,E1 -1887.222,E2 -1887.222} C_VEL
LIN {X 0,Y 580.041,Z 557.832,A -85,B 0,C 180,E1 -1888.612,E2 -1888.612} C_VEL
LIN {X 0,Y 580.036,Z 558.5,A -85,B 0,C 180,E1 -1890,E2 -1890} C_VEL
LIN {X 0,Y 580.041,Z 557.833,A -85,B 0,C 180,E1 -1891.389,E2 -1891.389} C_VEL
LIN {X 0,Y 580.041,Z 555.833,A -85,B 0,C 180,E1 -1892.778,E2 -1892.778} C_VEL
LIN {X 0,Y 580.102,Z 552.444,A -85,B 0,C 180,E1 -1894.168,E2 -1894.168} C_VEL
LIN {X 0,Y 580.128,Z 547.568,A -85,B 0,C 180,E1 -1895.562,E2 -1895.562} C_VEL
LIN {X 0,Y 580.141,Z 541.053,A -85,B 0,C 180,E1 -1896.958,E2 -1896.958} C_VEL
LIN {X 0,Y 580.192,Z 533.801,A -85,B 0,C 180,E1 -1898.183,E2 -1898.183} C_VEL
LIN {X 0,Y 580.283,Z 524.824,A -85,B 0,C 180,E1 -1899.41,E2 -1899.41} C_VEL
LIN {X 0,Y 580.356,Z 515.393,A -85,B 0,C 180,E1 -1900.466,E2 -1900.466} C_VEL
LIN {X 0,Y 580.475,Z 505.322,A -85,B 0,C 180,E1 -1901.404,E2 -1901.404} C_VEL
LIN {X 0,Y 580.617,Z 493.436,A -85,B 0,C 180,E1 -1902.318,E2 -1902.318} C_VEL
LIN {X 0,Y 580.73,Z 480.65,A -85,B 0,C 180,E1 -1903.115,E2 -1903.115} C_VEL
LIN {X 0,Y 580.897,Z 468.161,A -85,B 0,C 180,E1 -1903.735,E2 -1903.735} C_VEL
LIN {X 0,Y 581.024,Z 455.128,A -85,B 0,C 180,E1 -1904.238,E2 -1904.238} C_VEL
LIN {X 0,Y 581.111,Z 441.075,A -85,B 0,C 180,E1 -1904.633,E2 -1904.633} C_VEL
LIN {X 0,Y 581.162,Z 426.622,A -85,B 0,C 180,E1 -1904.89,E2 -1904.89} C_VEL
LIN {X 0,Y 581.324,Z 300.212,A -85,B 0,C 180,E1 -1906.475,E2 -1906.475} C_VEL
LIN {X 0,Y 580.594,Z 296.017,A -85,B 0,C 180,E1 -1906.572,E2 -1906.572} C_VEL
LIN {X 0,Y 580.694,Z 275.968,A -85,B 0,C 180,E1 -1909.263,E2 -1909.263} C_VEL
LIN {X 0,Y 580.946,Z 257.217,A -85,B 0,C 180,E1 -1911.838,E2 -1911.838} C_VEL
LIN {X 0,Y 580.909,Z 248.987,A -85,B 0,C 180,E1 -1912.989,E2 -1912.989} C_VEL
LIN {X 0,Y 580.336,Z 245.931,A -85,B 0,C 180,E1 -1913.487,E2 -1913.487} C_VEL
LIN {X 0,Y 580.291,Z 245.823,A -85,B 0,C 180,E1 -1916.334,E2 -1916.334} C_VEL
LIN {X 0,Y 580.3,Z 245.817,A -85,B 0,C 180,E1 -1919.309,E2 -1919.309} C_VEL
LIN {X 0,Y 580.299,Z 245.824,A -85,B 0,C 180,E1 -1922.2,E2 -1922.2} C_VEL
LIN {X 0,Y 580.288,Z 245.829,A -85,B 0,C 180,E1 -1924.696,E2 -1924.696} C_VEL
LIN {X 0,Y 580.295,Z 245.82,A -85,B 0,C 180,E1 -1927.268,E2 -1927.268} C_VEL
LIN {X 0,Y 580.289,Z 245.829,A -85,B 0,C 180,E1 -1930.27,E2 -1930.27} C_VEL
LIN {X 0,Y 580.279,Z 245.827,A -85,B 0,C 180,E1 -1932.705,E2 -1932.705} C_VEL
LIN {X 0,Y 580.265,Z 245.825,A -85,B 0,C 180,E1 -1935.608,E2 -1935.608} C_VEL
LIN {X 0,Y 580.3,Z 245.83,A -85,B 0,C 180,E1 -1938.233,E2 -1938.233} C_VEL
LIN {X 0,Y 580.286,Z 245.822,A -85,B 0,C 180,E1 -1940.966,E2 -1940.966} C_VEL
LIN {X 0,Y 580.291,Z 245.822,A -85,B 0,C 180,E1 -1943.598,E2 -1943.598} C_VEL
LIN {X 0,Y 580.313,Z 245.823,A -85,B 0,C 180,E1 -1946.145,E2 -1946.145} C_VEL
LIN {X 0,Y 580.282,Z 245.824,A -85,B 0,C 180,E1 -1948.615,E2 -1948.615} C_VEL
LIN {X 0,Y 580.287,Z 245.821,A -85,B 0,C 180,E1 -1951.024,E2 -1951.024} C_VEL
LIN {X 0,Y 580.32,Z 245.821,A -85,B 0,C 180,E1 -1953.658,E2 -1953.658} C_VEL
LIN {X 0,Y 580.275,Z 245.825,A -85,B 0,C 180,E1 -1956.442,E2 -1956.442} C_VEL
LIN {X 0,Y 580.268,Z 245.826,A -85,B 0,C 180,E1 -1959.437,E2 -1959.437} C_VEL
LIN {X 0,Y 580.274,Z 245.83,A -85,B 0,C 180,E1 -1961.645,E2 -1961.645} C_VEL
LIN {X 0,Y 580.276,Z 245.831,A -85,B 0,C 180,E1 -1963.826,E2 -1963.826} C_VEL
LIN {X 0,Y 580.319,Z 245.824,A -85,B 0,C 180,E1 -1965.983,E2 -1965.983} C_VEL
LIN {X 0,Y 580.295,Z 245.819,A -85,B 0,C 180,E1 -1968.827,E2 -1968.827} C_VEL
LIN {X 0,Y 580.327,Z 245.826,A -85,B 0,C 180,E1 -1971.644,E2 -1971.644} C_VEL
LIN {X 0,Y 580.32,Z 245.817,A -85,B 0,C 180,E1 -1974.44,E2 -1974.44} C_VEL
LIN {X 0,Y 580.337,Z 245.818,A -85,B 0,C 180,E1 -1977.224,E2 -1977.224} C_VEL
LIN {X 0,Y 580.344,Z 245.817,A -85,B 0,C 180,E1 -1980,E2 -1980} C_VEL
LIN {X 0,Y 580.338,Z 245.814,A -85,B 0,C 180,E1 -1982.777,E2 -1982.777} C_VEL
LIN {X 0,Y 580.32,Z 245.825,A -85,B 0,C 180,E1 -1985.56,E2 -1985.56} C_VEL
LIN {X 0,Y 580.327,Z 245.815,A -85,B 0,C 180,E1 -1988.356,E2 -1988.356} C_VEL
LIN {X 0,Y 580.29,Z 245.829,A -85,B 0,C 180,E1 -1991.191,E2 -1991.191} C_VEL
LIN {X 0,Y 580.319,Z 245.817,A -85,B 0,C 180,E1 -1994.017,E2 -1994.017} C_VEL
LIN {X 0,Y 580.306,Z 245.824,A -85,B 0,C 180,E1 -1996.915,E2 -1996.915} C_VEL
LIN {X 0,Y 580.3,Z 245.82,A -85,B 0,C 180,E1 -1999.823,E2 -1999.823} C_VEL
LIN {X 0,Y 580.274,Z 245.829,A -85,B 0,C 180,E1 -2001.34,E2 -2001.34} C_VEL
LIN {X 0,Y 579.579,Z 245.911,A -85,B 0,C 180,E1 -2001.919,E2 -2001.919} C_VEL
LIN {X 0,Y 576.704,Z 246.273,A -85,B 0,C 180,E1 -2002.859,E2 -2002.859} C_VEL
LIN {X 0,Y 574.31,Z 246.568,A -85,B 0,C 180,E1 -2003.615,E2 -2003.615} C_VEL
LIN {X 0,Y 573.311,Z 246.691,A -85,B 0,C 180,E1 -2004.199,E2 -2004.199} C_VEL
LIN {X 0,Y 573.244,Z 246.7,A -85,B 0,C 180,E1 -2004.396,E2 -2004.396} C_VEL
LIN {X 0,Y 573.248,Z 246.706,A -85,B 0,C 180,E1 -2006.976,E2 -2006.976} C_VEL
LIN {X 0,Y 573.246,Z 246.701,A -85,B 0,C 180,E1 -2009.49,E2 -2009.49} C_VEL
LIN {X 0,Y 573.249,Z 246.696,A -85,B 0,C 180,E1 -2012.23,E2 -2012.23} C_VEL
LIN {X 0,Y 573.247,Z 246.701,A -85,B 0,C 180,E1 -2014.775,E2 -2014.775} C_VEL
LIN {X 0,Y 573.249,Z 246.703,A -85,B 0,C 180,E1 -2017.167,E2 -2017.167} C_VEL
LIN {X 0,Y 573.244,Z 246.698,A -85,B 0,C 180,E1 -2019.608,E2 -2019.608} C_VEL
LIN {X 0,Y 573.236,Z 246.704,A -85,B 0,C 180,E1 -2022.642,E2 -2022.642} C_VEL
LIN {X 0,Y 573.236,Z 246.7,A -85,B 0,C 180,E1 -2025.668,E2 -2025.668} C_VEL
LIN {X 0,Y 573.242,Z 246.704,A -85,B 0,C 180,E1 -2028.545,E2 -2028.545} C_VEL
LIN {X 0,Y 573.242,Z 246.699,A -85,B 0,C 180,E1 -2031.299,E2 -2031.299} C_VEL
LIN {X 0,Y 573.243,Z 246.702,A -85,B 0,C 180,E1 -2034.015,E2 -2034.015} C_VEL
LIN {X 0,Y 573.285,Z 246.703,A -85,B 0,C 180,E1 -2036.52,E2 -2036.52} C_VEL
LIN {X 0,Y 573.228,Z 246.702,A -85,B 0,C 180,E1 -2039.118,E2 -2039.118} C_VEL
LIN {X 0,Y 573.238,Z 246.698,A -85,B 0,C 180,E1 -2041.436,E2 -2041.436} C_VEL
LIN {X 0,Y 573.266,Z 246.7,A -85,B 0,C 180,E1 -2043.811,E2 -2043.811} C_VEL
LIN {X 0,Y 573.232,Z 246.708,A -85,B 0,C 180,E1 -2046.135,E2 -2046.135} C_VEL
LIN {X 0,Y 573.288,Z 246.909,A -85,B 0,C 180,E1 -2047.475,E2 -2047.475} C_VEL
LIN {X 0,Y 573.969,Z 251.836,A -85,B 0,C 180,E1 -2048.26,E2 -2048.26} C_VEL
LIN {X 0,Y 573.695,Z 270.913,A -85,B 0,C 180,E1 -2051.057,E2 -2051.057} C_VEL
LIN {X 0,Y 573.577,Z 286.266,A -85,B 0,C 180,E1 -2053.257,E2 -2053.257} C_VEL
LIN {X 0,Y 574.036,Z 289.031,A -85,B 0,C 180,E1 -2053.339,E2 -2053.339} C_VEL
LIN {X 0,Y 574.571,Z 291.989,A -85,B 0,C 180,E1 -2053.393,E2 -2053.393} C_VEL
LIN {X 0,Y 574.28,Z 423.915,A -85,B 0,C 180,E1 -2055.086,E2 -2055.086} C_VEL
LIN {X 0,Y 574.173,Z 438.305,A -85,B 0,C 180,E1 -2055.42,E2 -2055.42} C_VEL
LIN {X 0,Y 574.03,Z 452.843,A -85,B 0,C 180,E1 -2055.917,E2 -2055.917} C_VEL
LIN {X 0,Y 573.848,Z 466.528,A -85,B 0,C 180,E1 -2056.544,E2 -2056.544} C_VEL
LIN {X 0,Y 573.687,Z 478.812,A -85,B 0,C 180,E1 -2057.261,E2 -2057.261} C_VEL
LIN {X 0,Y 573.55,Z 491.213,A -85,B 0,C 180,E1 -2058.156,E2 -2058.156} C_VEL
LIN {X 0,Y 573.438,Z 501.708,A -85,B 0,C 180,E1 -2059.082,E2 -2059.082} C_VEL
LIN {X 0,Y 573.245,Z 511.477,A -85,B 0,C 180,E1 -2060.117,E2 -2060.117} C_VEL
LIN {X 0,Y 573.202,Z 519.86,A -85,B 0,C 180,E1 -2061.184,E2 -2061.184} C_VEL
LIN {X 0,Y 573.111,Z 527.872,A -85,B 0,C 180,E1 -2062.425,E2 -2062.425} C_VEL
LIN {X 0,Y 573.022,Z 534.322,A -85,B 0,C 180,E1 -2063.663,E2 -2063.663} C_VEL
LIN {X 0,Y 573,Z 538.798,A -85,B 0,C 180,E1 -2064.722,E2 -2064.722} C_VEL
LIN {X 0,Y 573.029,Z 542.31,A -85,B 0,C 180,E1 -2065.78,E2 -2065.78} C_VEL
LIN {X 0,Y 572.957,Z 545.742,A -85,B 0,C 180,E1 -2067.188,E2 -2067.188} C_VEL
LIN {X 0,Y 572.944,Z 547.784,A -85,B 0,C 180,E1 -2068.594,E2 -2068.594} C_VEL
LIN {X 0,Y 572.937,Z 548.496,A -85,B 0,C 180,E1 -2070,E2 -2070} C_VEL
LIN {X 0,Y 572.942,Z 547.88,A -85,B 0,C 180,E1 -2071.406,E2 -2071.406} C_VEL
LIN {X 0,Y 572.954,Z 545.924,A -85,B 0,C 180,E1 -2072.812,E2 -2072.812} C_VEL
LIN {X 0,Y 573.03,Z 542.579,A -85,B 0,C 180,E1 -2074.22,E2 -2074.22} C_VEL
LIN {X 0,Y 573.056,Z 537.751,A -85,B 0,C 180,E1 -2075.63,E2 -2075.63} C_VEL
LIN {X 0,Y 573.054,Z 531.285,A -85,B 0,C 180,E1 -2077.044,E2 -2077.044} C_VEL
LIN {X 0,Y 573.142,Z 524.086,A -85,B 0,C 180,E1 -2078.284,E2 -2078.284} C_VEL
LIN {X 0,Y 573.225,Z 515.185,A -85,B 0,C 180,E1 -2079.527,E2 -2079.527} C_VEL
LIN {X 0,Y 573.35,Z 505.841,A -85,B 0,C 180,E1 -2080.595,E2 -2080.595} C_VEL
LIN {X 0,Y 573.476,Z 495.492,A -85,B 0,C 180,E1 -2081.576,E2 -2081.576} C_VEL
LIN {X 0,Y 573.626,Z 484.079,A -85,B 0,C 180,E1 -2082.47,E2 -2082.47} C_VEL
LIN {X 0,Y 573.802,Z 471.437,A -85,B 0,C 180,E1 -2083.276,E2 -2083.276} C_VEL
LIN {X 0,Y 573.973,Z 459.153,A -85,B 0,C 180,E1 -2083.904,E2 -2083.904} C_VEL
LIN {X 0,Y 574.152,Z 445.305,A -85,B 0,C 180,E1 -2084.451,E2 -2084.451} C_VEL
LIN {X 0,Y 574.224,Z 431.009,A -85,B 0,C 180,E1 -2084.859,E2 -2084.859} C_VEL
LIN {X 0,Y 574.324,Z 416.601,A -85,B 0,C 180,E1 -2085.117,E2 -2085.117} C_VEL
LIN {X 0,Y 574.478,Z 291.254,A -85,B 0,C 180,E1 -2086.709,E2 -2086.709} C_VEL
LIN {X 0,Y 573.599,Z 286.504,A -85,B 0,C 180,E1 -2086.815,E2 -2086.815} C_VEL
LIN {X 0,Y 573.749,Z 268.985,A -85,B 0,C 180,E1 -2089.313,E2 -2089.313} C_VEL
LIN {X 0,Y 573.985,Z 251.174,A -85,B 0,C 180,E1 -2091.928,E2 -2091.928} C_VEL
LIN {X 0,Y 573.306,Z 246.818,A -85,B 0,C 180,E1 -2092.643,E2 -2092.643} C_VEL
LIN {X 0,Y 573.256,Z 246.7,A -85,B 0,C 180,E1 -2095.409,E2 -2095.409} C_VEL
LIN {X 0,Y 573.253,Z 246.701,A -85,B 0,C 180,E1 -2098.029,E2 -2098.029} C_VEL
LIN {X 0,Y 573.245,Z 246.702,A -85,B 0,C 180,E1 -2100.175,E2 -2100.175} C_VEL
LIN {X 0,Y 573.254,Z 246.698,A -85,B 0,C 180,E1 -2102.644,E2 -2102.644} C_VEL
LIN {X 0,Y 573.252,Z 246.701,A -85,B 0,C 180,E1 -2105.184,E2 -2105.184} C_VEL
LIN {X 0,Y 573.233,Z 246.705,A -85,B 0,C 180,E1 -2107.807,E2 -2107.807} C_VEL
LIN {X 0,Y 573.267,Z 246.696,A -85,B 0,C 180,E1 -2110.527,E2 -2110.527} C_VEL
LIN {X 0,Y 573.248,Z 246.704,A -85,B 0,C 180,E1 -2113.669,E2 -2113.669} C_VEL
LIN {X 0,Y 573.234,Z 246.7,A -85,B 0,C 180,E1 -2116.64,E2 -2116.64} C_VEL
LIN {X 0,Y 573.269,Z 246.702,A -85,B 0,C 180,E1 -2119.477,E2 -2119.477} C_VEL
LIN {X 0,Y 573.231,Z 246.701,A -85,B 0,C 180,E1 -2122.192,E2 -2122.192} C_VEL
LIN {X 0,Y 573.264,Z 246.699,A -85,B 0,C 180,E1 -2124.816,E2 -2124.816} C_VEL
LIN {X 0,Y 573.249,Z 246.702,A -85,B 0,C 180,E1 -2127.354,E2 -2127.354} C_VEL
LIN {X 0,Y 573.25,Z 246.699,A -85,B 0,C 180,E1 -2129.824,E2 -2129.824} C_VEL
LIN {X 0,Y 573.281,Z 246.695,A -85,B 0,C 180,E1 -2132.235,E2 -2132.235} C_VEL
LIN {X 0,Y 573.267,Z 246.7,A -85,B 0,C 180,E1 -2135.366,E2 -2135.366} C_VEL
LIN {X 0,Y 573.221,Z 246.703,A -85,B 0,C 180,E1 -2138.419,E2 -2138.419} C_VEL
LIN {X 0,Y 573.269,Z 246.701,A -85,B 0,C 180,E1 -2140.728,E2 -2140.728} C_VEL
LIN {X 0,Y 573.251,Z 246.697,A -85,B 0,C 180,E1 -2143.622,E2 -2143.622} C_VEL
LIN {X 0,Y 573.233,Z 246.704,A -85,B 0,C 180,E1 -2146.529,E2 -2146.529} C_VEL
LIN {X 0,Y 573.274,Z 246.705,A -85,B 0,C 180,E1 -2148.734,E2 -2148.734} C_VEL
LIN {X 0,Y 573.283,Z 246.692,A -85,B 0,C 180,E1 -2151.54,E2 -2151.54} C_VEL
LIN {X 0,Y 573.287,Z 246.699,A -85,B 0,C 180,E1 -2154.372,E2 -2154.372} C_VEL
LIN {X 0,Y 573.3,Z 246.69,A -85,B 0,C 180,E1 -2157.892,E2 -2157.892} C_VEL
LIN {X 0,Y 573.329,Z 246.695,A -85,B 0,C 180,E1 -2160.702,E2 -2160.702} C_VEL
LIN {X 0,Y 573.233,Z 246.698,A -85,B 0,C 180,E1 -2163.514,E2 -2163.514} C_VEL
LIN {X 0,Y 573.286,Z 246.693,A -85,B 0,C 180,E1 -2165.628,E2 -2165.628} C_VEL
LIN {X 0,Y 573.298,Z 246.699,A -85,B 0,C 180,E1 -2168.459,E2 -2168.459} C_VEL
LIN {X 0,Y 573.261,Z 246.695,A -85,B 0,C 180,E1 -2171.312,E2 -2171.312} C_VEL
LIN {X 0,Y 573.265,Z 246.705,A -85,B 0,C 180,E1 -2174.193,E2 -2174.193} C_VEL
LIN {X 0,Y 573.251,Z 246.697,A -85,B 0,C 180,E1 -2177.112,E2 -2177.112} C_VEL
LIN {X 0,Y 573.246,Z 246.707,A -85,B 0,C 180,E1 -2180.077,E2 -2180.077} C_VEL
LIN {X 0,Y 573.225,Z 246.7,A -85,B 0,C 180,E1 -2183.1,E2 -2183.1} C_VEL
LIN {X 0,Y 573.247,Z 246.7,A -85,B 0,C 180,E1 -2185.41,E2 -2185.41} C_VEL
LIN {X 0,Y 573.256,Z 246.706,A -85,B 0,C 180,E1 -2188.032,E2 -2188.032} C_VEL
LIN {X 0,Y 573.237,Z 246.699,A -85,B 0,C 180,E1 -2190.886,E2 -2190.886} C_VEL
LIN {X 0,Y 573.254,Z 246.699,A -85,B 0,C 180,E1 -2193.525,E2 -2193.525} C_VEL
LIN {X 0,Y 573.255,Z 246.703,A -85,B 0,C 180,E1 -2196.049,E2 -2196.049} C_VEL
LIN {X 0,Y 573.244,Z 246.699,A -85,B 0,C 180,E1 -2198.701,E2 -2198.701} C_VEL
LIN {X 0,Y 573.248,Z 246.705,A -85,B 0,C 180,E1 -2201.596,E2 -2201.596} C_VEL
LIN {X 0,Y 573.23,Z 246.702,A -85,B 0,C 180,E1 -2204.334,E2 -2204.334} C_VEL
LIN {X 0,Y 573.246,Z 246.704,A -85,B 0,C 180,E1 -2207.358,E2 -2207.358} C_VEL
LIN {X 0,Y 573.243,Z 246.7,A -85,B 0,C 180,E1 -2210.394,E2 -2210.394} C_VEL
LIN {X 0,Y 573.249,Z 246.7,A -85,B 0,C 180,E1 -2213.078,E2 -2213.078} C_VEL
LIN {X 0,Y 573.269,Z 246.701,A -85,B 0,C 180,E1 -2215.672,E2 -2215.672} C_VEL
LIN {X 0,Y 573.247,Z 246.699,A -85,B 0,C 180,E1 -2218.186,E2 -2218.186} C_VEL
LIN {X 0,Y 573.263,Z 246.692,A -85,B 0,C 180,E1 -2220.635,E2 -2220.635} C_VEL
LIN {X 0,Y 573.25,Z 246.704,A -85,B 0,C 180,E1 -2223.025,E2 -2223.025} C_VEL
LIN {X 0,Y 573.275,Z 246.704,A -85,B 0,C 180,E1 -2225.367,E2 -2225.367} C_VEL
LIN {X 0,Y 573.304,Z 246.908,A -85,B 0,C 180,E1 -2226.38,E2 -2226.38} C_VEL
LIN {X 0,Y 574.11,Z 251.815,A -85,B 0,C 180,E1 -2227.129,E2 -2227.129} C_VEL
LIN {X 0,Y 573.858,Z 273.331,A -85,B 0,C 180,E1 -2230.133,E2 -2230.133} C_VEL
LIN {X 0,Y 573.588,Z 294.938,A -85,B 0,C 180,E1 -2233.1,E2 -2233.1} C_VEL
LIN {X 0,Y 573.663,Z 296.53,A -85,B 0,C 180,E1 -2233.246,E2 -2233.246} C_VEL
LIN {X 0,Y 574.585,Z 302.21,A -85,B 0,C 180,E1 -2233.351,E2 -2233.351} C_VEL
LIN {X 0,Y 574.298,Z 433.904,A -85,B 0,C 180,E1 -2235.041,E2 -2235.041} C_VEL
LIN {X 0,Y 574.183,Z 448.116,A -85,B 0,C 180,E1 -2235.37,E2 -2235.37} C_VEL
LIN {X 0,Y 574.019,Z 461.718,A -85,B 0,C 180,E1 -2235.826,E2 -2235.826} C_VEL
LIN {X 0,Y 573.889,Z 475.649,A -85,B 0,C 180,E1 -2236.455,E2 -2236.455} C_VEL
LIN {X 0,Y 573.711,Z 488.107,A -85,B 0,C 180,E1 -2237.172,E2 -2237.172} C_VEL
LIN {X 0,Y 573.531,Z 500.647,A -85,B 0,C 180,E1 -2238.066,E2 -2238.066} C_VEL
LIN {X 0,Y 573.449,Z 510.854,A -85,B 0,C 180,E1 -2238.955,E2 -2238.955} C_VEL
LIN {X 0,Y 573.269,Z 520.336,A -85,B 0,C 180,E1 -2239.939,E2 -2239.939} C_VEL
LIN {X 0,Y 573.19,Z 528.914,A -85,B 0,C 180,E1 -2241.006,E2 -2241.006} C_VEL
LIN {X 0,Y 573.111,Z 537.117,A -85,B 0,C 180,E1 -2242.248,E2 -2242.248} C_VEL
LIN {X 0,Y 573.036,Z 543.448,A -85,B 0,C 180,E1 -2243.427,E2 -2243.427} C_VEL
LIN {X 0,Y 573.001,Z 548.962,A -85,B 0,C 180,E1 -2244.722,E2 -2244.722} C_VEL
LIN {X 0,Y 573.028,Z 552.443,A -85,B 0,C 180,E1 -2245.78,E2 -2245.78} C_VEL
LIN {X 0,Y 572.956,Z 555.832,A -85,B 0,C 180,E1 -2247.188,E2 -2247.188} C_VEL
LIN {X 0,Y 572.941,Z 557.833,A -85,B 0,C 180,E1 -2248.594,E2 -2248.594} C_VEL
LIN {X 0,Y 572.937,Z 558.5,A -85,B 0,C 180,E1 -2250,E2 -2250} C_VEL
LIN {X 0,Y 572.941,Z 557.833,A -85,B 0,C 180,E1 -2251.406,E2 -2251.406} C_VEL
LIN {X 0,Y 572.956,Z 555.834,A -85,B 0,C 180,E1 -2252.812,E2 -2252.812} C_VEL
LIN {X 0,Y 573.028,Z 552.445,A -85,B 0,C 180,E1 -2254.22,E2 -2254.22} C_VEL
LIN {X 0,Y 573.057,Z 547.568,A -85,B 0,C 180,E1 -2255.63,E2 -2255.63} C_VEL
LIN {X 0,Y 573.065,Z 542.818,A -85,B 0,C 180,E1 -2256.699,E2 -2256.699} C_VEL
LIN {X 0,Y 573.126,Z 536.038,A -85,B 0,C 180,E1 -2257.929,E2 -2257.929} C_VEL
LIN {X 0,Y 573.225,Z 527.559,A -85,B 0,C 180,E1 -2259.171,E2 -2259.171} C_VEL
LIN {X 0,Y 573.304,Z 518.709,A -85,B 0,C 180,E1 -2260.239,E2 -2260.239} C_VEL
LIN {X 0,Y 573.462,Z 507.992,A -85,B 0,C 180,E1 -2261.308,E2 -2261.308} C_VEL
LIN {X 0,Y 573.62,Z 497.143,A -85,B 0,C 180,E1 -2262.201,E2 -2262.201} C_VEL
LIN {X 0,Y 573.738,Z 485.26,A -85,B 0,C 180,E1 -2263.008,E2 -2263.008} C_VEL
LIN {X 0,Y 573.946,Z 472.101,A -85,B 0,C 180,E1 -2263.724,E2 -2263.724} C_VEL
LIN {X 0,Y 574.095,Z 458.795,A -85,B 0,C 180,E1 -2264.285,E2 -2264.285} C_VEL
LIN {X 0,Y 574.212,Z 444.627,A -85,B 0,C 180,E1 -2264.724,E2 -2264.724} C_VEL
LIN {X 0,Y 574.314,Z 431.149,A -85,B 0,C 180,E1 -2265.004,E2 -2265.004} C_VEL
LIN {X 0,Y 574.504,Z 300.913,A -85,B 0,C 180,E1 -2266.668,E2 -2266.668} C_VEL
LIN {X 0,Y 573.639,Z 296.252,A -85,B 0,C 180,E1 -2266.766,E2 -2266.766} C_VEL
LIN {X 0,Y 573.577,Z 292.263,A -85,B 0,C 180,E1 -2267.267,E2 -2267.267} C_VEL
LIN {X 0,Y 573.871,Z 271.986,A -85,B 0,C 180,E1 -2270.054,E2 -2270.054} C_VEL
LIN {X 0,Y 574.125,Z 251.815,A -85,B 0,C 180,E1 -2272.871,E2 -2272.871} C_VEL
